  STRUCT
   STAT0 : ARRAY  [0 .. 999 ] OF BOOL ;
  END_STRUCT ;
BEGIN
   STAT0[0] := FALSE;
   STAT0[1] := FALSE;
   STAT0[2] := FALSE;
   STAT0[3] := FALSE;
   STAT0[4] := FALSE;
   STAT0[5] := FALSE;
   STAT0[6] := FALSE;
   STAT0[7] := FALSE;
   STAT0[8] := FALSE;
   STAT0[9] := FALSE;
   STAT0[10] := FALSE;
   STAT0[11] := FALSE;
   STAT0[12] := FALSE;
   STAT0[13] := FALSE;
   STAT0[14] := FALSE;
   STAT0[15] := FALSE;
   STAT0[16] := FALSE;
   STAT0[17] := FALSE;
   STAT0[18] := FALSE;
   STAT0[19] := FALSE;
   STAT0[20] := FALSE;
   STAT0[21] := FALSE;
   STAT0[22] := FALSE;
   STAT0[23] := FALSE;
   STAT0[24] := FALSE;
   STAT0[25] := FALSE;
   STAT0[26] := FALSE;
   STAT0[27] := FALSE;
   STAT0[28] := FALSE;
   STAT0[29] := FALSE;
   STAT0[30] := FALSE;
   STAT0[31] := FALSE;
   STAT0[32] := FALSE;
   STAT0[33] := FALSE;
   STAT0[34] := FALSE;
   STAT0[35] := FALSE;
   STAT0[36] := FALSE;
   STAT0[37] := FALSE;
   STAT0[38] := FALSE;
   STAT0[39] := FALSE;
   STAT0[40] := FALSE;
   STAT0[41] := FALSE;
   STAT0[42] := FALSE;
   STAT0[43] := FALSE;
   STAT0[44] := FALSE;
   STAT0[45] := FALSE;
   STAT0[46] := FALSE;
   STAT0[47] := FALSE;
   STAT0[48] := FALSE;
   STAT0[49] := FALSE;
   STAT0[50] := FALSE;
   STAT0[51] := FALSE;
   STAT0[52] := FALSE;
   STAT0[53] := FALSE;
   STAT0[54] := FALSE;
   STAT0[55] := FALSE;
   STAT0[56] := FALSE;
   STAT0[57] := FALSE;
   STAT0[58] := FALSE;
   STAT0[59] := FALSE;
   STAT0[60] := FALSE;
   STAT0[61] := FALSE;
   STAT0[62] := FALSE;
   STAT0[63] := FALSE;
   STAT0[64] := FALSE;
   STAT0[65] := FALSE;
   STAT0[66] := FALSE;
   STAT0[67] := FALSE;
   STAT0[68] := FALSE;
   STAT0[69] := FALSE;
   STAT0[70] := FALSE;
   STAT0[71] := FALSE;
   STAT0[72] := FALSE;
   STAT0[73] := FALSE;
   STAT0[74] := FALSE;
   STAT0[75] := FALSE;
   STAT0[76] := FALSE;
   STAT0[77] := FALSE;
   STAT0[78] := FALSE;
   STAT0[79] := FALSE;
   STAT0[80] := FALSE;
   STAT0[81] := FALSE;
   STAT0[82] := FALSE;
   STAT0[83] := FALSE;
   STAT0[84] := FALSE;
   STAT0[85] := FALSE;
   STAT0[86] := FALSE;
   STAT0[87] := FALSE;
   STAT0[88] := FALSE;
   STAT0[89] := FALSE;
   STAT0[90] := FALSE;
   STAT0[91] := FALSE;
   STAT0[92] := FALSE;
   STAT0[93] := FALSE;
   STAT0[94] := FALSE;
   STAT0[95] := FALSE;
   STAT0[96] := FALSE;
   STAT0[97] := FALSE;
   STAT0[98] := FALSE;
   STAT0[99] := FALSE;
   STAT0[100] := FALSE;
   STAT0[101] := FALSE;
   STAT0[102] := FALSE;
   STAT0[103] := FALSE;
   STAT0[104] := FALSE;
   STAT0[105] := FALSE;
   STAT0[106] := FALSE;
   STAT0[107] := FALSE;
   STAT0[108] := FALSE;
   STAT0[109] := FALSE;
   STAT0[110] := FALSE;
   STAT0[111] := FALSE;
   STAT0[112] := FALSE;
   STAT0[113] := FALSE;
   STAT0[114] := FALSE;
   STAT0[115] := FALSE;
   STAT0[116] := FALSE;
   STAT0[117] := FALSE;
   STAT0[118] := FALSE;
   STAT0[119] := FALSE;
   STAT0[120] := FALSE;
   STAT0[121] := FALSE;
   STAT0[122] := FALSE;
   STAT0[123] := FALSE;
   STAT0[124] := FALSE;
   STAT0[125] := FALSE;
   STAT0[126] := FALSE;
   STAT0[127] := FALSE;
   STAT0[128] := FALSE;
   STAT0[129] := FALSE;
   STAT0[130] := FALSE;
   STAT0[131] := FALSE;
   STAT0[132] := FALSE;
   STAT0[133] := FALSE;
   STAT0[134] := FALSE;
   STAT0[135] := FALSE;
   STAT0[136] := FALSE;
   STAT0[137] := FALSE;
   STAT0[138] := FALSE;
   STAT0[139] := FALSE;
   STAT0[140] := FALSE;
   STAT0[141] := FALSE;
   STAT0[142] := FALSE;
   STAT0[143] := FALSE;
   STAT0[144] := FALSE;
   STAT0[145] := FALSE;
   STAT0[146] := FALSE;
   STAT0[147] := FALSE;
   STAT0[148] := FALSE;
   STAT0[149] := FALSE;
   STAT0[150] := FALSE;
   STAT0[151] := FALSE;
   STAT0[152] := FALSE;
   STAT0[153] := FALSE;
   STAT0[154] := FALSE;
   STAT0[155] := FALSE;
   STAT0[156] := FALSE;
   STAT0[157] := FALSE;
   STAT0[158] := FALSE;
   STAT0[159] := FALSE;
   STAT0[160] := FALSE;
   STAT0[161] := FALSE;
   STAT0[162] := FALSE;
   STAT0[163] := FALSE;
   STAT0[164] := FALSE;
   STAT0[165] := FALSE;
   STAT0[166] := FALSE;
   STAT0[167] := FALSE;
   STAT0[168] := FALSE;
   STAT0[169] := FALSE;
   STAT0[170] := FALSE;
   STAT0[171] := FALSE;
   STAT0[172] := FALSE;
   STAT0[173] := FALSE;
   STAT0[174] := FALSE;
   STAT0[175] := FALSE;
   STAT0[176] := FALSE;
   STAT0[177] := FALSE;
   STAT0[178] := FALSE;
   STAT0[179] := FALSE;
   STAT0[180] := FALSE;
   STAT0[181] := FALSE;
   STAT0[182] := FALSE;
   STAT0[183] := FALSE;
   STAT0[184] := FALSE;
   STAT0[185] := FALSE;
   STAT0[186] := FALSE;
   STAT0[187] := FALSE;
   STAT0[188] := FALSE;
   STAT0[189] := FALSE;
   STAT0[190] := FALSE;
   STAT0[191] := FALSE;
   STAT0[192] := FALSE;
   STAT0[193] := FALSE;
   STAT0[194] := FALSE;
   STAT0[195] := FALSE;
   STAT0[196] := FALSE;
   STAT0[197] := FALSE;
   STAT0[198] := FALSE;
   STAT0[199] := FALSE;
   STAT0[200] := FALSE;
   STAT0[201] := FALSE;
   STAT0[202] := FALSE;
   STAT0[203] := FALSE;
   STAT0[204] := FALSE;
   STAT0[205] := FALSE;
   STAT0[206] := FALSE;
   STAT0[207] := FALSE;
   STAT0[208] := FALSE;
   STAT0[209] := FALSE;
   STAT0[210] := FALSE;
   STAT0[211] := FALSE;
   STAT0[212] := FALSE;
   STAT0[213] := FALSE;
   STAT0[214] := FALSE;
   STAT0[215] := FALSE;
   STAT0[216] := FALSE;
   STAT0[217] := FALSE;
   STAT0[218] := FALSE;
   STAT0[219] := FALSE;
   STAT0[220] := FALSE;
   STAT0[221] := FALSE;
   STAT0[222] := FALSE;
   STAT0[223] := FALSE;
   STAT0[224] := FALSE;
   STAT0[225] := FALSE;
   STAT0[226] := FALSE;
   STAT0[227] := FALSE;
   STAT0[228] := FALSE;
   STAT0[229] := FALSE;
   STAT0[230] := FALSE;
   STAT0[231] := FALSE;
   STAT0[232] := FALSE;
   STAT0[233] := FALSE;
   STAT0[234] := FALSE;
   STAT0[235] := FALSE;
   STAT0[236] := FALSE;
   STAT0[237] := FALSE;
   STAT0[238] := FALSE;
   STAT0[239] := FALSE;
   STAT0[240] := FALSE;
   STAT0[241] := FALSE;
   STAT0[242] := FALSE;
   STAT0[243] := FALSE;
   STAT0[244] := FALSE;
   STAT0[245] := FALSE;
   STAT0[246] := FALSE;
   STAT0[247] := FALSE;
   STAT0[248] := FALSE;
   STAT0[249] := FALSE;
   STAT0[250] := FALSE;
   STAT0[251] := FALSE;
   STAT0[252] := FALSE;
   STAT0[253] := FALSE;
   STAT0[254] := FALSE;
   STAT0[255] := FALSE;
   STAT0[256] := FALSE;
   STAT0[257] := FALSE;
   STAT0[258] := FALSE;
   STAT0[259] := FALSE;
   STAT0[260] := FALSE;
   STAT0[261] := FALSE;
   STAT0[262] := FALSE;
   STAT0[263] := FALSE;
   STAT0[264] := FALSE;
   STAT0[265] := FALSE;
   STAT0[266] := FALSE;
   STAT0[267] := FALSE;
   STAT0[268] := FALSE;
   STAT0[269] := FALSE;
   STAT0[270] := FALSE;
   STAT0[271] := FALSE;
   STAT0[272] := FALSE;
   STAT0[273] := FALSE;
   STAT0[274] := FALSE;
   STAT0[275] := FALSE;
   STAT0[276] := FALSE;
   STAT0[277] := FALSE;
   STAT0[278] := FALSE;
   STAT0[279] := FALSE;
   STAT0[280] := FALSE;
   STAT0[281] := FALSE;
   STAT0[282] := FALSE;
   STAT0[283] := FALSE;
   STAT0[284] := FALSE;
   STAT0[285] := FALSE;
   STAT0[286] := FALSE;
   STAT0[287] := FALSE;
   STAT0[288] := FALSE;
   STAT0[289] := FALSE;
   STAT0[290] := FALSE;
   STAT0[291] := FALSE;
   STAT0[292] := FALSE;
   STAT0[293] := FALSE;
   STAT0[294] := FALSE;
   STAT0[295] := FALSE;
   STAT0[296] := FALSE;
   STAT0[297] := FALSE;
   STAT0[298] := FALSE;
   STAT0[299] := FALSE;
   STAT0[300] := FALSE;
   STAT0[301] := FALSE;
   STAT0[302] := FALSE;
   STAT0[303] := FALSE;
   STAT0[304] := FALSE;
   STAT0[305] := FALSE;
   STAT0[306] := FALSE;
   STAT0[307] := FALSE;
   STAT0[308] := FALSE;
   STAT0[309] := FALSE;
   STAT0[310] := FALSE;
   STAT0[311] := FALSE;
   STAT0[312] := FALSE;
   STAT0[313] := FALSE;
   STAT0[314] := FALSE;
   STAT0[315] := FALSE;
   STAT0[316] := FALSE;
   STAT0[317] := FALSE;
   STAT0[318] := FALSE;
   STAT0[319] := FALSE;
   STAT0[320] := FALSE;
   STAT0[321] := FALSE;
   STAT0[322] := FALSE;
   STAT0[323] := FALSE;
   STAT0[324] := FALSE;
   STAT0[325] := FALSE;
   STAT0[326] := FALSE;
   STAT0[327] := FALSE;
   STAT0[328] := FALSE;
   STAT0[329] := FALSE;
   STAT0[330] := FALSE;
   STAT0[331] := FALSE;
   STAT0[332] := FALSE;
   STAT0[333] := FALSE;
   STAT0[334] := FALSE;
   STAT0[335] := FALSE;
   STAT0[336] := FALSE;
   STAT0[337] := FALSE;
   STAT0[338] := FALSE;
   STAT0[339] := FALSE;
   STAT0[340] := FALSE;
   STAT0[341] := FALSE;
   STAT0[342] := FALSE;
   STAT0[343] := FALSE;
   STAT0[344] := FALSE;
   STAT0[345] := FALSE;
   STAT0[346] := FALSE;
   STAT0[347] := FALSE;
   STAT0[348] := FALSE;
   STAT0[349] := FALSE;
   STAT0[350] := FALSE;
   STAT0[351] := FALSE;
   STAT0[352] := FALSE;
   STAT0[353] := FALSE;
   STAT0[354] := FALSE;
   STAT0[355] := FALSE;
   STAT0[356] := FALSE;
   STAT0[357] := FALSE;
   STAT0[358] := FALSE;
   STAT0[359] := FALSE;
   STAT0[360] := FALSE;
   STAT0[361] := FALSE;
   STAT0[362] := FALSE;
   STAT0[363] := FALSE;
   STAT0[364] := FALSE;
   STAT0[365] := FALSE;
   STAT0[366] := FALSE;
   STAT0[367] := FALSE;
   STAT0[368] := FALSE;
   STAT0[369] := FALSE;
   STAT0[370] := FALSE;
   STAT0[371] := FALSE;
   STAT0[372] := FALSE;
   STAT0[373] := FALSE;
   STAT0[374] := FALSE;
   STAT0[375] := FALSE;
   STAT0[376] := FALSE;
   STAT0[377] := FALSE;
   STAT0[378] := FALSE;
   STAT0[379] := FALSE;
   STAT0[380] := FALSE;
   STAT0[381] := FALSE;
   STAT0[382] := FALSE;
   STAT0[383] := FALSE;
   STAT0[384] := FALSE;
   STAT0[385] := FALSE;
   STAT0[386] := FALSE;
   STAT0[387] := FALSE;
   STAT0[388] := FALSE;
   STAT0[389] := FALSE;
   STAT0[390] := FALSE;
   STAT0[391] := FALSE;
   STAT0[392] := FALSE;
   STAT0[393] := FALSE;
   STAT0[394] := FALSE;
   STAT0[395] := FALSE;
   STAT0[396] := FALSE;
   STAT0[397] := FALSE;
   STAT0[398] := FALSE;
   STAT0[399] := FALSE;
   STAT0[400] := FALSE;
   STAT0[401] := FALSE;
   STAT0[402] := FALSE;
   STAT0[403] := FALSE;
   STAT0[404] := FALSE;
   STAT0[405] := FALSE;
   STAT0[406] := FALSE;
   STAT0[407] := FALSE;
   STAT0[408] := FALSE;
   STAT0[409] := FALSE;
   STAT0[410] := FALSE;
   STAT0[411] := FALSE;
   STAT0[412] := FALSE;
   STAT0[413] := FALSE;
   STAT0[414] := FALSE;
   STAT0[415] := FALSE;
   STAT0[416] := FALSE;
   STAT0[417] := FALSE;
   STAT0[418] := FALSE;
   STAT0[419] := FALSE;
   STAT0[420] := FALSE;
   STAT0[421] := FALSE;
   STAT0[422] := FALSE;
   STAT0[423] := FALSE;
   STAT0[424] := FALSE;
   STAT0[425] := FALSE;
   STAT0[426] := FALSE;
   STAT0[427] := FALSE;
   STAT0[428] := FALSE;
   STAT0[429] := FALSE;
   STAT0[430] := FALSE;
   STAT0[431] := FALSE;
   STAT0[432] := FALSE;
   STAT0[433] := FALSE;
   STAT0[434] := FALSE;
   STAT0[435] := FALSE;
   STAT0[436] := FALSE;
   STAT0[437] := FALSE;
   STAT0[438] := FALSE;
   STAT0[439] := FALSE;
   STAT0[440] := FALSE;
   STAT0[441] := FALSE;
   STAT0[442] := FALSE;
   STAT0[443] := FALSE;
   STAT0[444] := FALSE;
   STAT0[445] := FALSE;
   STAT0[446] := FALSE;
   STAT0[447] := FALSE;
   STAT0[448] := FALSE;
   STAT0[449] := FALSE;
   STAT0[450] := FALSE;
   STAT0[451] := FALSE;
   STAT0[452] := FALSE;
   STAT0[453] := FALSE;
   STAT0[454] := FALSE;
   STAT0[455] := FALSE;
   STAT0[456] := FALSE;
   STAT0[457] := FALSE;
   STAT0[458] := FALSE;
   STAT0[459] := FALSE;
   STAT0[460] := FALSE;
   STAT0[461] := FALSE;
   STAT0[462] := FALSE;
   STAT0[463] := FALSE;
   STAT0[464] := FALSE;
   STAT0[465] := FALSE;
   STAT0[466] := FALSE;
   STAT0[467] := FALSE;
   STAT0[468] := FALSE;
   STAT0[469] := FALSE;
   STAT0[470] := FALSE;
   STAT0[471] := FALSE;
   STAT0[472] := FALSE;
   STAT0[473] := FALSE;
   STAT0[474] := FALSE;
   STAT0[475] := FALSE;
   STAT0[476] := FALSE;
   STAT0[477] := FALSE;
   STAT0[478] := FALSE;
   STAT0[479] := FALSE;
   STAT0[480] := FALSE;
   STAT0[481] := FALSE;
   STAT0[482] := FALSE;
   STAT0[483] := FALSE;
   STAT0[484] := FALSE;
   STAT0[485] := FALSE;
   STAT0[486] := FALSE;
   STAT0[487] := FALSE;
   STAT0[488] := FALSE;
   STAT0[489] := FALSE;
   STAT0[490] := FALSE;
   STAT0[491] := FALSE;
   STAT0[492] := FALSE;
   STAT0[493] := FALSE;
   STAT0[494] := FALSE;
   STAT0[495] := FALSE;
   STAT0[496] := FALSE;
   STAT0[497] := FALSE;
   STAT0[498] := FALSE;
   STAT0[499] := FALSE;
   STAT0[500] := FALSE;
   STAT0[501] := FALSE;
   STAT0[502] := FALSE;
   STAT0[503] := FALSE;
   STAT0[504] := FALSE;
   STAT0[505] := FALSE;
   STAT0[506] := FALSE;
   STAT0[507] := FALSE;
   STAT0[508] := FALSE;
   STAT0[509] := FALSE;
   STAT0[510] := FALSE;
   STAT0[511] := FALSE;
   STAT0[512] := FALSE;
   STAT0[513] := FALSE;
   STAT0[514] := FALSE;
   STAT0[515] := FALSE;
   STAT0[516] := FALSE;
   STAT0[517] := FALSE;
   STAT0[518] := FALSE;
   STAT0[519] := FALSE;
   STAT0[520] := FALSE;
   STAT0[521] := FALSE;
   STAT0[522] := FALSE;
   STAT0[523] := FALSE;
   STAT0[524] := FALSE;
   STAT0[525] := FALSE;
   STAT0[526] := FALSE;
   STAT0[527] := FALSE;
   STAT0[528] := FALSE;
   STAT0[529] := FALSE;
   STAT0[530] := FALSE;
   STAT0[531] := FALSE;
   STAT0[532] := FALSE;
   STAT0[533] := FALSE;
   STAT0[534] := FALSE;
   STAT0[535] := FALSE;
   STAT0[536] := FALSE;
   STAT0[537] := FALSE;
   STAT0[538] := FALSE;
   STAT0[539] := FALSE;
   STAT0[540] := FALSE;
   STAT0[541] := FALSE;
   STAT0[542] := FALSE;
   STAT0[543] := FALSE;
   STAT0[544] := FALSE;
   STAT0[545] := FALSE;
   STAT0[546] := FALSE;
   STAT0[547] := FALSE;
   STAT0[548] := FALSE;
   STAT0[549] := FALSE;
   STAT0[550] := FALSE;
   STAT0[551] := FALSE;
   STAT0[552] := FALSE;
   STAT0[553] := FALSE;
   STAT0[554] := FALSE;
   STAT0[555] := FALSE;
   STAT0[556] := FALSE;
   STAT0[557] := FALSE;
   STAT0[558] := FALSE;
   STAT0[559] := FALSE;
   STAT0[560] := FALSE;
   STAT0[561] := FALSE;
   STAT0[562] := FALSE;
   STAT0[563] := FALSE;
   STAT0[564] := FALSE;
   STAT0[565] := FALSE;
   STAT0[566] := FALSE;
   STAT0[567] := FALSE;
   STAT0[568] := FALSE;
   STAT0[569] := FALSE;
   STAT0[570] := FALSE;
   STAT0[571] := FALSE;
   STAT0[572] := FALSE;
   STAT0[573] := FALSE;
   STAT0[574] := FALSE;
   STAT0[575] := FALSE;
   STAT0[576] := FALSE;
   STAT0[577] := FALSE;
   STAT0[578] := FALSE;
   STAT0[579] := FALSE;
   STAT0[580] := FALSE;
   STAT0[581] := FALSE;
   STAT0[582] := FALSE;
   STAT0[583] := FALSE;
   STAT0[584] := FALSE;
   STAT0[585] := FALSE;
   STAT0[586] := FALSE;
   STAT0[587] := FALSE;
   STAT0[588] := FALSE;
   STAT0[589] := FALSE;
   STAT0[590] := FALSE;
   STAT0[591] := FALSE;
   STAT0[592] := FALSE;
   STAT0[593] := FALSE;
   STAT0[594] := FALSE;
   STAT0[595] := FALSE;
   STAT0[596] := FALSE;
   STAT0[597] := FALSE;
   STAT0[598] := FALSE;
   STAT0[599] := FALSE;
   STAT0[600] := FALSE;
   STAT0[601] := FALSE;
   STAT0[602] := FALSE;
   STAT0[603] := FALSE;
   STAT0[604] := FALSE;
   STAT0[605] := FALSE;
   STAT0[606] := FALSE;
   STAT0[607] := FALSE;
   STAT0[608] := FALSE;
   STAT0[609] := FALSE;
   STAT0[610] := FALSE;
   STAT0[611] := FALSE;
   STAT0[612] := FALSE;
   STAT0[613] := FALSE;
   STAT0[614] := FALSE;
   STAT0[615] := FALSE;
   STAT0[616] := FALSE;
   STAT0[617] := FALSE;
   STAT0[618] := FALSE;
   STAT0[619] := FALSE;
   STAT0[620] := FALSE;
   STAT0[621] := FALSE;
   STAT0[622] := FALSE;
   STAT0[623] := FALSE;
   STAT0[624] := FALSE;
   STAT0[625] := FALSE;
   STAT0[626] := FALSE;
   STAT0[627] := FALSE;
   STAT0[628] := FALSE;
   STAT0[629] := FALSE;
   STAT0[630] := FALSE;
   STAT0[631] := FALSE;
   STAT0[632] := FALSE;
   STAT0[633] := FALSE;
   STAT0[634] := FALSE;
   STAT0[635] := FALSE;
   STAT0[636] := FALSE;
   STAT0[637] := FALSE;
   STAT0[638] := FALSE;
   STAT0[639] := FALSE;
   STAT0[640] := FALSE;
   STAT0[641] := FALSE;
   STAT0[642] := FALSE;
   STAT0[643] := FALSE;
   STAT0[644] := FALSE;
   STAT0[645] := FALSE;
   STAT0[646] := FALSE;
   STAT0[647] := FALSE;
   STAT0[648] := FALSE;
   STAT0[649] := FALSE;
   STAT0[650] := FALSE;
   STAT0[651] := FALSE;
   STAT0[652] := FALSE;
   STAT0[653] := FALSE;
   STAT0[654] := FALSE;
   STAT0[655] := FALSE;
   STAT0[656] := FALSE;
   STAT0[657] := FALSE;
   STAT0[658] := FALSE;
   STAT0[659] := FALSE;
   STAT0[660] := FALSE;
   STAT0[661] := FALSE;
   STAT0[662] := FALSE;
   STAT0[663] := FALSE;
   STAT0[664] := FALSE;
   STAT0[665] := FALSE;
   STAT0[666] := FALSE;
   STAT0[667] := FALSE;
   STAT0[668] := FALSE;
   STAT0[669] := FALSE;
   STAT0[670] := FALSE;
   STAT0[671] := FALSE;
   STAT0[672] := FALSE;
   STAT0[673] := FALSE;
   STAT0[674] := FALSE;
   STAT0[675] := FALSE;
   STAT0[676] := FALSE;
   STAT0[677] := FALSE;
   STAT0[678] := FALSE;
   STAT0[679] := FALSE;
   STAT0[680] := FALSE;
   STAT0[681] := FALSE;
   STAT0[682] := FALSE;
   STAT0[683] := FALSE;
   STAT0[684] := FALSE;
   STAT0[685] := FALSE;
   STAT0[686] := FALSE;
   STAT0[687] := FALSE;
   STAT0[688] := FALSE;
   STAT0[689] := FALSE;
   STAT0[690] := FALSE;
   STAT0[691] := FALSE;
   STAT0[692] := FALSE;
   STAT0[693] := FALSE;
   STAT0[694] := FALSE;
   STAT0[695] := FALSE;
   STAT0[696] := FALSE;
   STAT0[697] := FALSE;
   STAT0[698] := FALSE;
   STAT0[699] := FALSE;
   STAT0[700] := FALSE;
   STAT0[701] := FALSE;
   STAT0[702] := FALSE;
   STAT0[703] := FALSE;
   STAT0[704] := FALSE;
   STAT0[705] := FALSE;
   STAT0[706] := FALSE;
   STAT0[707] := FALSE;
   STAT0[708] := FALSE;
   STAT0[709] := FALSE;
   STAT0[710] := FALSE;
   STAT0[711] := FALSE;
   STAT0[712] := FALSE;
   STAT0[713] := FALSE;
   STAT0[714] := FALSE;
   STAT0[715] := FALSE;
   STAT0[716] := FALSE;
   STAT0[717] := FALSE;
   STAT0[718] := FALSE;
   STAT0[719] := FALSE;
   STAT0[720] := FALSE;
   STAT0[721] := FALSE;
   STAT0[722] := FALSE;
   STAT0[723] := FALSE;
   STAT0[724] := FALSE;
   STAT0[725] := FALSE;
   STAT0[726] := FALSE;
   STAT0[727] := FALSE;
   STAT0[728] := FALSE;
   STAT0[729] := FALSE;
   STAT0[730] := FALSE;
   STAT0[731] := FALSE;
   STAT0[732] := FALSE;
   STAT0[733] := FALSE;
   STAT0[734] := FALSE;
   STAT0[735] := FALSE;
   STAT0[736] := FALSE;
   STAT0[737] := FALSE;
   STAT0[738] := FALSE;
   STAT0[739] := FALSE;
   STAT0[740] := FALSE;
   STAT0[741] := FALSE;
   STAT0[742] := FALSE;
   STAT0[743] := FALSE;
   STAT0[744] := FALSE;
   STAT0[745] := FALSE;
   STAT0[746] := FALSE;
   STAT0[747] := FALSE;
   STAT0[748] := FALSE;
   STAT0[749] := FALSE;
   STAT0[750] := FALSE;
   STAT0[751] := FALSE;
   STAT0[752] := FALSE;
   STAT0[753] := FALSE;
   STAT0[754] := FALSE;
   STAT0[755] := FALSE;
   STAT0[756] := FALSE;
   STAT0[757] := FALSE;
   STAT0[758] := FALSE;
   STAT0[759] := FALSE;
   STAT0[760] := FALSE;
   STAT0[761] := FALSE;
   STAT0[762] := FALSE;
   STAT0[763] := FALSE;
   STAT0[764] := FALSE;
   STAT0[765] := FALSE;
   STAT0[766] := FALSE;
   STAT0[767] := FALSE;
   STAT0[768] := FALSE;
   STAT0[769] := FALSE;
   STAT0[770] := FALSE;
   STAT0[771] := FALSE;
   STAT0[772] := FALSE;
   STAT0[773] := FALSE;
   STAT0[774] := FALSE;
   STAT0[775] := FALSE;
   STAT0[776] := FALSE;
   STAT0[777] := FALSE;
   STAT0[778] := FALSE;
   STAT0[779] := FALSE;
   STAT0[780] := FALSE;
   STAT0[781] := FALSE;
   STAT0[782] := FALSE;
   STAT0[783] := FALSE;
   STAT0[784] := FALSE;
   STAT0[785] := FALSE;
   STAT0[786] := FALSE;
   STAT0[787] := FALSE;
   STAT0[788] := FALSE;
   STAT0[789] := FALSE;
   STAT0[790] := FALSE;
   STAT0[791] := FALSE;
   STAT0[792] := FALSE;
   STAT0[793] := FALSE;
   STAT0[794] := FALSE;
   STAT0[795] := FALSE;
   STAT0[796] := FALSE;
   STAT0[797] := FALSE;
   STAT0[798] := FALSE;
   STAT0[799] := FALSE;
   STAT0[800] := FALSE;
   STAT0[801] := FALSE;
   STAT0[802] := FALSE;
   STAT0[803] := FALSE;
   STAT0[804] := FALSE;
   STAT0[805] := FALSE;
   STAT0[806] := FALSE;
   STAT0[807] := FALSE;
   STAT0[808] := FALSE;
   STAT0[809] := FALSE;
   STAT0[810] := FALSE;
   STAT0[811] := FALSE;
   STAT0[812] := FALSE;
   STAT0[813] := FALSE;
   STAT0[814] := FALSE;
   STAT0[815] := FALSE;
   STAT0[816] := FALSE;
   STAT0[817] := FALSE;
   STAT0[818] := FALSE;
   STAT0[819] := FALSE;
   STAT0[820] := FALSE;
   STAT0[821] := FALSE;
   STAT0[822] := FALSE;
   STAT0[823] := FALSE;
   STAT0[824] := FALSE;
   STAT0[825] := FALSE;
   STAT0[826] := FALSE;
   STAT0[827] := FALSE;
   STAT0[828] := FALSE;
   STAT0[829] := FALSE;
   STAT0[830] := FALSE;
   STAT0[831] := FALSE;
   STAT0[832] := FALSE;
   STAT0[833] := FALSE;
   STAT0[834] := FALSE;
   STAT0[835] := FALSE;
   STAT0[836] := FALSE;
   STAT0[837] := FALSE;
   STAT0[838] := FALSE;
   STAT0[839] := FALSE;
   STAT0[840] := FALSE;
   STAT0[841] := FALSE;
   STAT0[842] := FALSE;
   STAT0[843] := FALSE;
   STAT0[844] := FALSE;
   STAT0[845] := FALSE;
   STAT0[846] := FALSE;
   STAT0[847] := FALSE;
   STAT0[848] := FALSE;
   STAT0[849] := FALSE;
   STAT0[850] := FALSE;
   STAT0[851] := FALSE;
   STAT0[852] := FALSE;
   STAT0[853] := FALSE;
   STAT0[854] := FALSE;
   STAT0[855] := FALSE;
   STAT0[856] := FALSE;
   STAT0[857] := FALSE;
   STAT0[858] := FALSE;
   STAT0[859] := FALSE;
   STAT0[860] := FALSE;
   STAT0[861] := FALSE;
   STAT0[862] := FALSE;
   STAT0[863] := FALSE;
   STAT0[864] := FALSE;
   STAT0[865] := FALSE;
   STAT0[866] := FALSE;
   STAT0[867] := FALSE;
   STAT0[868] := FALSE;
   STAT0[869] := FALSE;
   STAT0[870] := FALSE;
   STAT0[871] := FALSE;
   STAT0[872] := FALSE;
   STAT0[873] := FALSE;
   STAT0[874] := FALSE;
   STAT0[875] := FALSE;
   STAT0[876] := FALSE;
   STAT0[877] := FALSE;
   STAT0[878] := FALSE;
   STAT0[879] := FALSE;
   STAT0[880] := FALSE;
   STAT0[881] := FALSE;
   STAT0[882] := FALSE;
   STAT0[883] := FALSE;
   STAT0[884] := FALSE;
   STAT0[885] := FALSE;
   STAT0[886] := FALSE;
   STAT0[887] := FALSE;
   STAT0[888] := FALSE;
   STAT0[889] := FALSE;
   STAT0[890] := FALSE;
   STAT0[891] := FALSE;
   STAT0[892] := FALSE;
   STAT0[893] := FALSE;
   STAT0[894] := FALSE;
   STAT0[895] := FALSE;
   STAT0[896] := FALSE;
   STAT0[897] := FALSE;
   STAT0[898] := FALSE;
   STAT0[899] := FALSE;
   STAT0[900] := FALSE;
   STAT0[901] := FALSE;
   STAT0[902] := FALSE;
   STAT0[903] := FALSE;
   STAT0[904] := FALSE;
   STAT0[905] := FALSE;
   STAT0[906] := FALSE;
   STAT0[907] := FALSE;
   STAT0[908] := FALSE;
   STAT0[909] := FALSE;
   STAT0[910] := FALSE;
   STAT0[911] := FALSE;
   STAT0[912] := FALSE;
   STAT0[913] := FALSE;
   STAT0[914] := FALSE;
   STAT0[915] := FALSE;
   STAT0[916] := FALSE;
   STAT0[917] := FALSE;
   STAT0[918] := FALSE;
   STAT0[919] := FALSE;
   STAT0[920] := FALSE;
   STAT0[921] := FALSE;
   STAT0[922] := FALSE;
   STAT0[923] := FALSE;
   STAT0[924] := FALSE;
   STAT0[925] := FALSE;
   STAT0[926] := FALSE;
   STAT0[927] := FALSE;
   STAT0[928] := FALSE;
   STAT0[929] := FALSE;
   STAT0[930] := FALSE;
   STAT0[931] := FALSE;
   STAT0[932] := FALSE;
   STAT0[933] := FALSE;
   STAT0[934] := FALSE;
   STAT0[935] := FALSE;
   STAT0[936] := FALSE;
   STAT0[937] := FALSE;
   STAT0[938] := FALSE;
   STAT0[939] := FALSE;
   STAT0[940] := FALSE;
   STAT0[941] := FALSE;
   STAT0[942] := FALSE;
   STAT0[943] := FALSE;
   STAT0[944] := FALSE;
   STAT0[945] := FALSE;
   STAT0[946] := FALSE;
   STAT0[947] := FALSE;
   STAT0[948] := FALSE;
   STAT0[949] := FALSE;
   STAT0[950] := FALSE;
   STAT0[951] := FALSE;
   STAT0[952] := FALSE;
   STAT0[953] := FALSE;
   STAT0[954] := FALSE;
   STAT0[955] := FALSE;
   STAT0[956] := FALSE;
   STAT0[957] := FALSE;
   STAT0[958] := FALSE;
   STAT0[959] := FALSE;
   STAT0[960] := FALSE;
   STAT0[961] := FALSE;
   STAT0[962] := FALSE;
   STAT0[963] := FALSE;
   STAT0[964] := FALSE;
   STAT0[965] := FALSE;
   STAT0[966] := FALSE;
   STAT0[967] := FALSE;
   STAT0[968] := FALSE;
   STAT0[969] := FALSE;
   STAT0[970] := FALSE;
   STAT0[971] := FALSE;
   STAT0[972] := FALSE;
   STAT0[973] := FALSE;
   STAT0[974] := FALSE;
   STAT0[975] := FALSE;
   STAT0[976] := FALSE;
   STAT0[977] := FALSE;
   STAT0[978] := FALSE;
   STAT0[979] := FALSE;
   STAT0[980] := FALSE;
   STAT0[981] := FALSE;
   STAT0[982] := FALSE;
   STAT0[983] := FALSE;
   STAT0[984] := FALSE;
   STAT0[985] := FALSE;
   STAT0[986] := FALSE;
   STAT0[987] := FALSE;
   STAT0[988] := FALSE;
   STAT0[989] := FALSE;
   STAT0[990] := FALSE;
   STAT0[991] := FALSE;
   STAT0[992] := FALSE;
   STAT0[993] := FALSE;
   STAT0[994] := FALSE;
   STAT0[995] := FALSE;
   STAT0[996] := FALSE;
   STAT0[997] := FALSE;
   STAT0[998] := FALSE;
   STAT0[999] := FALSE;
END_DATA_BLOCK

DATA_BLOCK DB 325
TITLE =
VERSION : 0.1


  STRUCT
   DP_DIAG1 : ARRAY  [1 .. 100 ] OF BYTE ;
   DP_DIAG2 : ARRAY  [1 .. 100 ] OF BYTE ;
   DP_DIAG3 : ARRAY  [1 .. 100 ] OF BYTE ;
   DP_DIAG4 : ARRAY  [1 .. 100 ] OF BYTE ;
   DP_DIAG5 : ARRAY  [1 .. 100 ] OF BYTE ;
   DP_DIAG6 : ARRAY  [1 .. 100 ] OF BYTE ;
   DP_DIAG7 : ARRAY  [1 .. 100 ] OF BYTE ;
   DP_DIAG8 : ARRAY  [1 .. 100 ] OF BYTE ;
   DP_DIAG9 : ARRAY  [1 .. 100 ] OF BYTE ;
   DP_DIAG10 : ARRAY  [1 .. 100 ] OF BYTE ;
  END_STRUCT ;
BEGIN
   DP_DIAG1[1] := B#16#FC;
   DP_DIAG1[2] := B#16#0;
   DP_DIAG1[3] := B#16#8;
   DP_DIAG1[4] := B#16#40;
   DP_DIAG1[5] := B#16#0;
   DP_DIAG1[6] := B#16#0;
   DP_DIAG1[7] := B#16#0;
   DP_DIAG1[8] := B#16#0;
   DP_DIAG1[9] := B#16#0;
   DP_DIAG1[10] := B#16#0;
   DP_DIAG1[11] := B#16#0;
   DP_DIAG1[12] := B#16#0;
   DP_DIAG1[13] := B#16#0;
   DP_DIAG1[14] := B#16#0;
   DP_DIAG1[15] := B#16#0;
   DP_DIAG1[16] := B#16#0;
   DP_DIAG1[17] := B#16#FC;
   DP_DIAG1[18] := B#16#0;
   DP_DIAG1[19] := B#16#8;
   DP_DIAG1[20] := B#16#40;
   DP_DIAG1[21] := B#16#0;
   DP_DIAG1[22] := B#16#0;
   DP_DIAG1[23] := B#16#0;
   DP_DIAG1[24] := B#16#0;
   DP_DIAG1[25] := B#16#0;
   DP_DIAG1[26] := B#16#0;
   DP_DIAG1[27] := B#16#0;
   DP_DIAG1[28] := B#16#0;
   DP_DIAG1[29] := B#16#0;
   DP_DIAG1[30] := B#16#0;
   DP_DIAG1[31] := B#16#0;
   DP_DIAG1[32] := B#16#0;
   DP_DIAG1[33] := B#16#4;
   DP_DIAG1[34] := B#16#0;
   DP_DIAG1[35] := B#16#0;
   DP_DIAG1[36] := B#16#0;
   DP_DIAG1[37] := B#16#0;
   DP_DIAG1[38] := B#16#0;
   DP_DIAG1[39] := B#16#0;
   DP_DIAG1[40] := B#16#0;
   DP_DIAG1[41] := B#16#0;
   DP_DIAG1[42] := B#16#0;
   DP_DIAG1[43] := B#16#0;
   DP_DIAG1[44] := B#16#0;
   DP_DIAG1[45] := B#16#0;
   DP_DIAG1[46] := B#16#0;
   DP_DIAG1[47] := B#16#0;
   DP_DIAG1[48] := B#16#0;
   DP_DIAG1[49] := B#16#0;
   DP_DIAG1[50] := B#16#0;
   DP_DIAG1[51] := B#16#0;
   DP_DIAG1[52] := B#16#0;
   DP_DIAG1[53] := B#16#0;
   DP_DIAG1[54] := B#16#0;
   DP_DIAG1[55] := B#16#0;
   DP_DIAG1[56] := B#16#0;
   DP_DIAG1[57] := B#16#0;
   DP_DIAG1[58] := B#16#0;
   DP_DIAG1[59] := B#16#0;
   DP_DIAG1[60] := B#16#0;
   DP_DIAG1[61] := B#16#0;
   DP_DIAG1[62] := B#16#0;
   DP_DIAG1[63] := B#16#0;
   DP_DIAG1[64] := B#16#0;
   DP_DIAG1[65] := B#16#0;
   DP_DIAG1[66] := B#16#0;
   DP_DIAG1[67] := B#16#4;
   DP_DIAG1[68] := B#16#0;
   DP_DIAG1[69] := B#16#0;
   DP_DIAG1[70] := B#16#0;
   DP_DIAG1[71] := B#16#0;
   DP_DIAG1[72] := B#16#0;
   DP_DIAG1[73] := B#16#0;
   DP_DIAG1[74] := B#16#0;
   DP_DIAG1[75] := B#16#0;
   DP_DIAG1[76] := B#16#0;
   DP_DIAG1[77] := B#16#0;
   DP_DIAG1[78] := B#16#0;
   DP_DIAG1[79] := B#16#0;
   DP_DIAG1[80] := B#16#0;
   DP_DIAG1[81] := B#16#0;
   DP_DIAG1[82] := B#16#0;
   DP_DIAG1[83] := B#16#0;
   DP_DIAG1[84] := B#16#1;
   DP_DIAG1[85] := B#16#0;
   DP_DIAG1[86] := B#16#0;
   DP_DIAG1[87] := B#16#0;
   DP_DIAG1[88] := B#16#0;
   DP_DIAG1[89] := B#16#0;
   DP_DIAG1[90] := B#16#0;
   DP_DIAG1[91] := B#16#0;
   DP_DIAG1[92] := B#16#0;
   DP_DIAG1[93] := B#16#0;
   DP_DIAG1[94] := B#16#0;
   DP_DIAG1[95] := B#16#0;
   DP_DIAG1[96] := B#16#0;
   DP_DIAG1[97] := B#16#0;
   DP_DIAG1[98] := B#16#0;
   DP_DIAG1[99] := B#16#0;
   DP_DIAG1[100] := B#16#0;
   DP_DIAG2[1] := B#16#0;
   DP_DIAG2[2] := B#16#0;
   DP_DIAG2[3] := B#16#0;
   DP_DIAG2[4] := B#16#0;
   DP_DIAG2[5] := B#16#0;
   DP_DIAG2[6] := B#16#0;
   DP_DIAG2[7] := B#16#0;
   DP_DIAG2[8] := B#16#0;
   DP_DIAG2[9] := B#16#0;
   DP_DIAG2[10] := B#16#0;
   DP_DIAG2[11] := B#16#0;
   DP_DIAG2[12] := B#16#0;
   DP_DIAG2[13] := B#16#0;
   DP_DIAG2[14] := B#16#0;
   DP_DIAG2[15] := B#16#0;
   DP_DIAG2[16] := B#16#0;
   DP_DIAG2[17] := B#16#0;
   DP_DIAG2[18] := B#16#0;
   DP_DIAG2[19] := B#16#0;
   DP_DIAG2[20] := B#16#0;
   DP_DIAG2[21] := B#16#0;
   DP_DIAG2[22] := B#16#0;
   DP_DIAG2[23] := B#16#0;
   DP_DIAG2[24] := B#16#0;
   DP_DIAG2[25] := B#16#0;
   DP_DIAG2[26] := B#16#0;
   DP_DIAG2[27] := B#16#0;
   DP_DIAG2[28] := B#16#0;
   DP_DIAG2[29] := B#16#0;
   DP_DIAG2[30] := B#16#0;
   DP_DIAG2[31] := B#16#0;
   DP_DIAG2[32] := B#16#0;
   DP_DIAG2[33] := B#16#0;
   DP_DIAG2[34] := B#16#0;
   DP_DIAG2[35] := B#16#0;
   DP_DIAG2[36] := B#16#0;
   DP_DIAG2[37] := B#16#0;
   DP_DIAG2[38] := B#16#0;
   DP_DIAG2[39] := B#16#0;
   DP_DIAG2[40] := B#16#0;
   DP_DIAG2[41] := B#16#0;
   DP_DIAG2[42] := B#16#0;
   DP_DIAG2[43] := B#16#0;
   DP_DIAG2[44] := B#16#0;
   DP_DIAG2[45] := B#16#0;
   DP_DIAG2[46] := B#16#0;
   DP_DIAG2[47] := B#16#0;
   DP_DIAG2[48] := B#16#0;
   DP_DIAG2[49] := B#16#0;
   DP_DIAG2[50] := B#16#0;
   DP_DIAG2[51] := B#16#0;
   DP_DIAG2[52] := B#16#0;
   DP_DIAG2[53] := B#16#0;
   DP_DIAG2[54] := B#16#0;
   DP_DIAG2[55] := B#16#0;
   DP_DIAG2[56] := B#16#0;
   DP_DIAG2[57] := B#16#0;
   DP_DIAG2[58] := B#16#0;
   DP_DIAG2[59] := B#16#0;
   DP_DIAG2[60] := B#16#0;
   DP_DIAG2[61] := B#16#0;
   DP_DIAG2[62] := B#16#0;
   DP_DIAG2[63] := B#16#0;
   DP_DIAG2[64] := B#16#0;
   DP_DIAG2[65] := B#16#0;
   DP_DIAG2[66] := B#16#0;
   DP_DIAG2[67] := B#16#0;
   DP_DIAG2[68] := B#16#0;
   DP_DIAG2[69] := B#16#0;
   DP_DIAG2[70] := B#16#0;
   DP_DIAG2[71] := B#16#0;
   DP_DIAG2[72] := B#16#0;
   DP_DIAG2[73] := B#16#0;
   DP_DIAG2[74] := B#16#0;
   DP_DIAG2[75] := B#16#0;
   DP_DIAG2[76] := B#16#0;
   DP_DIAG2[77] := B#16#0;
   DP_DIAG2[78] := B#16#0;
   DP_DIAG2[79] := B#16#0;
   DP_DIAG2[80] := B#16#0;
   DP_DIAG2[81] := B#16#0;
   DP_DIAG2[82] := B#16#0;
   DP_DIAG2[83] := B#16#0;
   DP_DIAG2[84] := B#16#0;
   DP_DIAG2[85] := B#16#0;
   DP_DIAG2[86] := B#16#0;
   DP_DIAG2[87] := B#16#0;
   DP_DIAG2[88] := B#16#0;
   DP_DIAG2[89] := B#16#0;
   DP_DIAG2[90] := B#16#0;
   DP_DIAG2[91] := B#16#0;
   DP_DIAG2[92] := B#16#0;
   DP_DIAG2[93] := B#16#0;
   DP_DIAG2[94] := B#16#0;
   DP_DIAG2[95] := B#16#0;
   DP_DIAG2[96] := B#16#0;
   DP_DIAG2[97] := B#16#0;
   DP_DIAG2[98] := B#16#0;
   DP_DIAG2[99] := B#16#0;
   DP_DIAG2[100] := B#16#0;
   DP_DIAG3[1] := B#16#0;
   DP_DIAG3[2] := B#16#0;
   DP_DIAG3[3] := B#16#0;
   DP_DIAG3[4] := B#16#0;
   DP_DIAG3[5] := B#16#0;
   DP_DIAG3[6] := B#16#0;
   DP_DIAG3[7] := B#16#0;
   DP_DIAG3[8] := B#16#0;
   DP_DIAG3[9] := B#16#0;
   DP_DIAG3[10] := B#16#0;
   DP_DIAG3[11] := B#16#0;
   DP_DIAG3[12] := B#16#0;
   DP_DIAG3[13] := B#16#0;
   DP_DIAG3[14] := B#16#0;
   DP_DIAG3[15] := B#16#0;
   DP_DIAG3[16] := B#16#0;
   DP_DIAG3[17] := B#16#0;
   DP_DIAG3[18] := B#16#0;
   DP_DIAG3[19] := B#16#0;
   DP_DIAG3[20] := B#16#0;
   DP_DIAG3[21] := B#16#0;
   DP_DIAG3[22] := B#16#0;
   DP_DIAG3[23] := B#16#0;
   DP_DIAG3[24] := B#16#0;
   DP_DIAG3[25] := B#16#0;
   DP_DIAG3[26] := B#16#0;
   DP_DIAG3[27] := B#16#0;
   DP_DIAG3[28] := B#16#0;
   DP_DIAG3[29] := B#16#0;
   DP_DIAG3[30] := B#16#0;
   DP_DIAG3[31] := B#16#0;
   DP_DIAG3[32] := B#16#0;
   DP_DIAG3[33] := B#16#0;
   DP_DIAG3[34] := B#16#0;
   DP_DIAG3[35] := B#16#0;
   DP_DIAG3[36] := B#16#0;
   DP_DIAG3[37] := B#16#0;
   DP_DIAG3[38] := B#16#0;
   DP_DIAG3[39] := B#16#0;
   DP_DIAG3[40] := B#16#0;
   DP_DIAG3[41] := B#16#0;
   DP_DIAG3[42] := B#16#0;
   DP_DIAG3[43] := B#16#0;
   DP_DIAG3[44] := B#16#0;
   DP_DIAG3[45] := B#16#0;
   DP_DIAG3[46] := B#16#0;
   DP_DIAG3[47] := B#16#0;
   DP_DIAG3[48] := B#16#0;
   DP_DIAG3[49] := B#16#0;
   DP_DIAG3[50] := B#16#0;
   DP_DIAG3[51] := B#16#0;
   DP_DIAG3[52] := B#16#0;
   DP_DIAG3[53] := B#16#0;
   DP_DIAG3[54] := B#16#0;
   DP_DIAG3[55] := B#16#0;
   DP_DIAG3[56] := B#16#0;
   DP_DIAG3[57] := B#16#0;
   DP_DIAG3[58] := B#16#0;
   DP_DIAG3[59] := B#16#0;
   DP_DIAG3[60] := B#16#0;
   DP_DIAG3[61] := B#16#0;
   DP_DIAG3[62] := B#16#0;
   DP_DIAG3[63] := B#16#0;
   DP_DIAG3[64] := B#16#0;
   DP_DIAG3[65] := B#16#0;
   DP_DIAG3[66] := B#16#0;
   DP_DIAG3[67] := B#16#0;
   DP_DIAG3[68] := B#16#0;
   DP_DIAG3[69] := B#16#0;
   DP_DIAG3[70] := B#16#0;
   DP_DIAG3[71] := B#16#0;
   DP_DIAG3[72] := B#16#0;
   DP_DIAG3[73] := B#16#0;
   DP_DIAG3[74] := B#16#0;
   DP_DIAG3[75] := B#16#0;
   DP_DIAG3[76] := B#16#0;
   DP_DIAG3[77] := B#16#0;
   DP_DIAG3[78] := B#16#0;
   DP_DIAG3[79] := B#16#0;
   DP_DIAG3[80] := B#16#0;
   DP_DIAG3[81] := B#16#0;
   DP_DIAG3[82] := B#16#0;
   DP_DIAG3[83] := B#16#0;
   DP_DIAG3[84] := B#16#0;
   DP_DIAG3[85] := B#16#0;
   DP_DIAG3[86] := B#16#0;
   DP_DIAG3[87] := B#16#0;
   DP_DIAG3[88] := B#16#0;
   DP_DIAG3[89] := B#16#0;
   DP_DIAG3[90] := B#16#0;
   DP_DIAG3[91] := B#16#0;
   DP_DIAG3[92] := B#16#0;
   DP_DIAG3[93] := B#16#0;
   DP_DIAG3[94] := B#16#0;
   DP_DIAG3[95] := B#16#0;
   DP_DIAG3[96] := B#16#0;
   DP_DIAG3[97] := B#16#0;
   DP_DIAG3[98] := B#16#0;
   DP_DIAG3[99] := B#16#0;
   DP_DIAG3[100] := B#16#0;
   DP_DIAG4[1] := B#16#0;
   DP_DIAG4[2] := B#16#0;
   DP_DIAG4[3] := B#16#0;
   DP_DIAG4[4] := B#16#0;
   DP_DIAG4[5] := B#16#0;
   DP_DIAG4[6] := B#16#0;
   DP_DIAG4[7] := B#16#0;
   DP_DIAG4[8] := B#16#0;
   DP_DIAG4[9] := B#16#0;
   DP_DIAG4[10] := B#16#0;
   DP_DIAG4[11] := B#16#0;
   DP_DIAG4[12] := B#16#0;
   DP_DIAG4[13] := B#16#0;
   DP_DIAG4[14] := B#16#0;
   DP_DIAG4[15] := B#16#0;
   DP_DIAG4[16] := B#16#0;
   DP_DIAG4[17] := B#16#0;
   DP_DIAG4[18] := B#16#0;
   DP_DIAG4[19] := B#16#0;
   DP_DIAG4[20] := B#16#0;
   DP_DIAG4[21] := B#16#0;
   DP_DIAG4[22] := B#16#0;
   DP_DIAG4[23] := B#16#0;
   DP_DIAG4[24] := B#16#0;
   DP_DIAG4[25] := B#16#0;
   DP_DIAG4[26] := B#16#0;
   DP_DIAG4[27] := B#16#0;
   DP_DIAG4[28] := B#16#0;
   DP_DIAG4[29] := B#16#0;
   DP_DIAG4[30] := B#16#0;
   DP_DIAG4[31] := B#16#0;
   DP_DIAG4[32] := B#16#0;
   DP_DIAG4[33] := B#16#0;
   DP_DIAG4[34] := B#16#0;
   DP_DIAG4[35] := B#16#0;
   DP_DIAG4[36] := B#16#0;
   DP_DIAG4[37] := B#16#0;
   DP_DIAG4[38] := B#16#0;
   DP_DIAG4[39] := B#16#0;
   DP_DIAG4[40] := B#16#0;
   DP_DIAG4[41] := B#16#0;
   DP_DIAG4[42] := B#16#0;
   DP_DIAG4[43] := B#16#0;
   DP_DIAG4[44] := B#16#0;
   DP_DIAG4[45] := B#16#0;
   DP_DIAG4[46] := B#16#0;
   DP_DIAG4[47] := B#16#0;
   DP_DIAG4[48] := B#16#0;
   DP_DIAG4[49] := B#16#0;
   DP_DIAG4[50] := B#16#0;
   DP_DIAG4[51] := B#16#0;
   DP_DIAG4[52] := B#16#0;
   DP_DIAG4[53] := B#16#0;
   DP_DIAG4[54] := B#16#0;
   DP_DIAG4[55] := B#16#0;
   DP_DIAG4[56] := B#16#0;
   DP_DIAG4[57] := B#16#0;
   DP_DIAG4[58] := B#16#0;
   DP_DIAG4[59] := B#16#0;
   DP_DIAG4[60] := B#16#0;
   DP_DIAG4[61] := B#16#0;
   DP_DIAG4[62] := B#16#0;
   DP_DIAG4[63] := B#16#0;
   DP_DIAG4[64] := B#16#0;
   DP_DIAG4[65] := B#16#0;
   DP_DIAG4[66] := B#16#0;
   DP_DIAG4[67] := B#16#0;
   DP_DIAG4[68] := B#16#0;
   DP_DIAG4[69] := B#16#0;
   DP_DIAG4[70] := B#16#0;
   DP_DIAG4[71] := B#16#0;
   DP_DIAG4[72] := B#16#0;
   DP_DIAG4[73] := B#16#0;
   DP_DIAG4[74] := B#16#0;
   DP_DIAG4[75] := B#16#0;
   DP_DIAG4[76] := B#16#0;
   DP_DIAG4[77] := B#16#0;
   DP_DIAG4[78] := B#16#0;
   DP_DIAG4[79] := B#16#0;
   DP_DIAG4[80] := B#16#0;
   DP_DIAG4[81] := B#16#0;
   DP_DIAG4[82] := B#16#0;
   DP_DIAG4[83] := B#16#0;
   DP_DIAG4[84] := B#16#0;
   DP_DIAG4[85] := B#16#0;
   DP_DIAG4[86] := B#16#0;
   DP_DIAG4[87] := B#16#0;
   DP_DIAG4[88] := B#16#0;
   DP_DIAG4[89] := B#16#0;
   DP_DIAG4[90] := B#16#0;
   DP_DIAG4[91] := B#16#0;
   DP_DIAG4[92] := B#16#0;
   DP_DIAG4[93] := B#16#0;
   DP_DIAG4[94] := B#16#0;
   DP_DIAG4[95] := B#16#0;
   DP_DIAG4[96] := B#16#0;
   DP_DIAG4[97] := B#16#0;
   DP_DIAG4[98] := B#16#0;
   DP_DIAG4[99] := B#16#0;
   DP_DIAG4[100] := B#16#0;
   DP_DIAG5[1] := B#16#0;
   DP_DIAG5[2] := B#16#0;
   DP_DIAG5[3] := B#16#0;
   DP_DIAG5[4] := B#16#0;
   DP_DIAG5[5] := B#16#0;
   DP_DIAG5[6] := B#16#0;
   DP_DIAG5[7] := B#16#0;
   DP_DIAG5[8] := B#16#0;
   DP_DIAG5[9] := B#16#0;
   DP_DIAG5[10] := B#16#0;
   DP_DIAG5[11] := B#16#0;
   DP_DIAG5[12] := B#16#0;
   DP_DIAG5[13] := B#16#0;
   DP_DIAG5[14] := B#16#0;
   DP_DIAG5[15] := B#16#0;
   DP_DIAG5[16] := B#16#0;
   DP_DIAG5[17] := B#16#0;
   DP_DIAG5[18] := B#16#0;
   DP_DIAG5[19] := B#16#0;
   DP_DIAG5[20] := B#16#0;
   DP_DIAG5[21] := B#16#0;
   DP_DIAG5[22] := B#16#0;
   DP_DIAG5[23] := B#16#0;
   DP_DIAG5[24] := B#16#0;
   DP_DIAG5[25] := B#16#0;
   DP_DIAG5[26] := B#16#0;
   DP_DIAG5[27] := B#16#0;
   DP_DIAG5[28] := B#16#0;
   DP_DIAG5[29] := B#16#0;
   DP_DIAG5[30] := B#16#0;
   DP_DIAG5[31] := B#16#0;
   DP_DIAG5[32] := B#16#0;
   DP_DIAG5[33] := B#16#0;
   DP_DIAG5[34] := B#16#0;
   DP_DIAG5[35] := B#16#0;
   DP_DIAG5[36] := B#16#0;
   DP_DIAG5[37] := B#16#0;
   DP_DIAG5[38] := B#16#0;
   DP_DIAG5[39] := B#16#0;
   DP_DIAG5[40] := B#16#0;
   DP_DIAG5[41] := B#16#0;
   DP_DIAG5[42] := B#16#0;
   DP_DIAG5[43] := B#16#0;
   DP_DIAG5[44] := B#16#0;
   DP_DIAG5[45] := B#16#0;
   DP_DIAG5[46] := B#16#0;
   DP_DIAG5[47] := B#16#0;
   DP_DIAG5[48] := B#16#0;
   DP_DIAG5[49] := B#16#0;
   DP_DIAG5[50] := B#16#0;
   DP_DIAG5[51] := B#16#0;
   DP_DIAG5[52] := B#16#0;
   DP_DIAG5[53] := B#16#0;
   DP_DIAG5[54] := B#16#0;
   DP_DIAG5[55] := B#16#0;
   DP_DIAG5[56] := B#16#0;
   DP_DIAG5[57] := B#16#0;
   DP_DIAG5[58] := B#16#0;
   DP_DIAG5[59] := B#16#0;
   DP_DIAG5[60] := B#16#0;
   DP_DIAG5[61] := B#16#0;
   DP_DIAG5[62] := B#16#0;
   DP_DIAG5[63] := B#16#0;
   DP_DIAG5[64] := B#16#0;
   DP_DIAG5[65] := B#16#0;
   DP_DIAG5[66] := B#16#0;
   DP_DIAG5[67] := B#16#0;
   DP_DIAG5[68] := B#16#0;
   DP_DIAG5[69] := B#16#0;
   DP_DIAG5[70] := B#16#0;
   DP_DIAG5[71] := B#16#0;
   DP_DIAG5[72] := B#16#0;
   DP_DIAG5[73] := B#16#0;
   DP_DIAG5[74] := B#16#0;
   DP_DIAG5[75] := B#16#0;
   DP_DIAG5[76] := B#16#0;
   DP_DIAG5[77] := B#16#0;
   DP_DIAG5[78] := B#16#0;
   DP_DIAG5[79] := B#16#0;
   DP_DIAG5[80] := B#16#0;
   DP_DIAG5[81] := B#16#0;
   DP_DIAG5[82] := B#16#0;
   DP_DIAG5[83] := B#16#0;
   DP_DIAG5[84] := B#16#0;
   DP_DIAG5[85] := B#16#0;
   DP_DIAG5[86] := B#16#0;
   DP_DIAG5[87] := B#16#0;
   DP_DIAG5[88] := B#16#0;
   DP_DIAG5[89] := B#16#0;
   DP_DIAG5[90] := B#16#0;
   DP_DIAG5[91] := B#16#0;
   DP_DIAG5[92] := B#16#0;
   DP_DIAG5[93] := B#16#0;
   DP_DIAG5[94] := B#16#0;
   DP_DIAG5[95] := B#16#0;
   DP_DIAG5[96] := B#16#0;
   DP_DIAG5[97] := B#16#0;
   DP_DIAG5[98] := B#16#0;
   DP_DIAG5[99] := B#16#0;
   DP_DIAG5[100] := B#16#0;
   DP_DIAG6[1] := B#16#0;
   DP_DIAG6[2] := B#16#0;
   DP_DIAG6[3] := B#16#0;
   DP_DIAG6[4] := B#16#0;
   DP_DIAG6[5] := B#16#0;
   DP_DIAG6[6] := B#16#0;
   DP_DIAG6[7] := B#16#0;
   DP_DIAG6[8] := B#16#0;
   DP_DIAG6[9] := B#16#0;
   DP_DIAG6[10] := B#16#0;
   DP_DIAG6[11] := B#16#0;
   DP_DIAG6[12] := B#16#0;
   DP_DIAG6[13] := B#16#0;
   DP_DIAG6[14] := B#16#0;
   DP_DIAG6[15] := B#16#0;
   DP_DIAG6[16] := B#16#0;
   DP_DIAG6[17] := B#16#0;
   DP_DIAG6[18] := B#16#0;
   DP_DIAG6[19] := B#16#0;
   DP_DIAG6[20] := B#16#0;
   DP_DIAG6[21] := B#16#0;
   DP_DIAG6[22] := B#16#0;
   DP_DIAG6[23] := B#16#0;
   DP_DIAG6[24] := B#16#0;
   DP_DIAG6[25] := B#16#0;
   DP_DIAG6[26] := B#16#0;
   DP_DIAG6[27] := B#16#0;
   DP_DIAG6[28] := B#16#0;
   DP_DIAG6[29] := B#16#0;
   DP_DIAG6[30] := B#16#0;
   DP_DIAG6[31] := B#16#0;
   DP_DIAG6[32] := B#16#0;
   DP_DIAG6[33] := B#16#0;
   DP_DIAG6[34] := B#16#0;
   DP_DIAG6[35] := B#16#0;
   DP_DIAG6[36] := B#16#0;
   DP_DIAG6[37] := B#16#0;
   DP_DIAG6[38] := B#16#0;
   DP_DIAG6[39] := B#16#0;
   DP_DIAG6[40] := B#16#0;
   DP_DIAG6[41] := B#16#0;
   DP_DIAG6[42] := B#16#0;
   DP_DIAG6[43] := B#16#0;
   DP_DIAG6[44] := B#16#0;
   DP_DIAG6[45] := B#16#0;
   DP_DIAG6[46] := B#16#0;
   DP_DIAG6[47] := B#16#0;
   DP_DIAG6[48] := B#16#0;
   DP_DIAG6[49] := B#16#0;
   DP_DIAG6[50] := B#16#0;
   DP_DIAG6[51] := B#16#0;
   DP_DIAG6[52] := B#16#0;
   DP_DIAG6[53] := B#16#0;
   DP_DIAG6[54] := B#16#0;
   DP_DIAG6[55] := B#16#0;
   DP_DIAG6[56] := B#16#0;
   DP_DIAG6[57] := B#16#0;
   DP_DIAG6[58] := B#16#0;
   DP_DIAG6[59] := B#16#0;
   DP_DIAG6[60] := B#16#0;
   DP_DIAG6[61] := B#16#0;
   DP_DIAG6[62] := B#16#0;
   DP_DIAG6[63] := B#16#0;
   DP_DIAG6[64] := B#16#0;
   DP_DIAG6[65] := B#16#0;
   DP_DIAG6[66] := B#16#0;
   DP_DIAG6[67] := B#16#0;
   DP_DIAG6[68] := B#16#0;
   DP_DIAG6[69] := B#16#0;
   DP_DIAG6[70] := B#16#0;
   DP_DIAG6[71] := B#16#0;
   DP_DIAG6[72] := B#16#0;
   DP_DIAG6[73] := B#16#0;
   DP_DIAG6[74] := B#16#0;
   DP_DIAG6[75] := B#16#0;
   DP_DIAG6[76] := B#16#0;
   DP_DIAG6[77] := B#16#0;
   DP_DIAG6[78] := B#16#0;
   DP_DIAG6[79] := B#16#0;
   DP_DIAG6[80] := B#16#0;
   DP_DIAG6[81] := B#16#0;
   DP_DIAG6[82] := B#16#0;
   DP_DIAG6[83] := B#16#0;
   DP_DIAG6[84] := B#16#0;
   DP_DIAG6[85] := B#16#0;
   DP_DIAG6[86] := B#16#0;
   DP_DIAG6[87] := B#16#0;
   DP_DIAG6[88] := B#16#0;
   DP_DIAG6[89] := B#16#0;
   DP_DIAG6[90] := B#16#0;
   DP_DIAG6[91] := B#16#0;
   DP_DIAG6[92] := B#16#0;
   DP_DIAG6[93] := B#16#0;
   DP_DIAG6[94] := B#16#0;
   DP_DIAG6[95] := B#16#0;
   DP_DIAG6[96] := B#16#0;
   DP_DIAG6[97] := B#16#0;
   DP_DIAG6[98] := B#16#0;
   DP_DIAG6[99] := B#16#0;
   DP_DIAG6[100] := B#16#0;
   DP_DIAG7[1] := B#16#0;
   DP_DIAG7[2] := B#16#0;
   DP_DIAG7[3] := B#16#0;
   DP_DIAG7[4] := B#16#0;
   DP_DIAG7[5] := B#16#0;
   DP_DIAG7[6] := B#16#0;
   DP_DIAG7[7] := B#16#0;
   DP_DIAG7[8] := B#16#0;
   DP_DIAG7[9] := B#16#0;
   DP_DIAG7[10] := B#16#0;
   DP_DIAG7[11] := B#16#0;
   DP_DIAG7[12] := B#16#0;
   DP_DIAG7[13] := B#16#0;
   DP_DIAG7[14] := B#16#0;
   DP_DIAG7[15] := B#16#0;
   DP_DIAG7[16] := B#16#0;
   DP_DIAG7[17] := B#16#0;
   DP_DIAG7[18] := B#16#0;
   DP_DIAG7[19] := B#16#0;
   DP_DIAG7[20] := B#16#0;
   DP_DIAG7[21] := B#16#0;
   DP_DIAG7[22] := B#16#0;
   DP_DIAG7[23] := B#16#0;
   DP_DIAG7[24] := B#16#0;
   DP_DIAG7[25] := B#16#0;
   DP_DIAG7[26] := B#16#0;
   DP_DIAG7[27] := B#16#0;
   DP_DIAG7[28] := B#16#0;
   DP_DIAG7[29] := B#16#0;
   DP_DIAG7[30] := B#16#0;
   DP_DIAG7[31] := B#16#0;
   DP_DIAG7[32] := B#16#0;
   DP_DIAG7[33] := B#16#0;
   DP_DIAG7[34] := B#16#0;
   DP_DIAG7[35] := B#16#0;
   DP_DIAG7[36] := B#16#0;
   DP_DIAG7[37] := B#16#0;
   DP_DIAG7[38] := B#16#0;
   DP_DIAG7[39] := B#16#0;
   DP_DIAG7[40] := B#16#0;
   DP_DIAG7[41] := B#16#0;
   DP_DIAG7[42] := B#16#0;
   DP_DIAG7[43] := B#16#0;
   DP_DIAG7[44] := B#16#0;
   DP_DIAG7[45] := B#16#0;
   DP_DIAG7[46] := B#16#0;
   DP_DIAG7[47] := B#16#0;
   DP_DIAG7[48] := B#16#0;
   DP_DIAG7[49] := B#16#0;
   DP_DIAG7[50] := B#16#0;
   DP_DIAG7[51] := B#16#0;
   DP_DIAG7[52] := B#16#0;
   DP_DIAG7[53] := B#16#0;
   DP_DIAG7[54] := B#16#0;
   DP_DIAG7[55] := B#16#0;
   DP_DIAG7[56] := B#16#0;
   DP_DIAG7[57] := B#16#0;
   DP_DIAG7[58] := B#16#0;
   DP_DIAG7[59] := B#16#0;
   DP_DIAG7[60] := B#16#0;
   DP_DIAG7[61] := B#16#0;
   DP_DIAG7[62] := B#16#0;
   DP_DIAG7[63] := B#16#0;
   DP_DIAG7[64] := B#16#0;
   DP_DIAG7[65] := B#16#0;
   DP_DIAG7[66] := B#16#0;
   DP_DIAG7[67] := B#16#0;
   DP_DIAG7[68] := B#16#0;
   DP_DIAG7[69] := B#16#0;
   DP_DIAG7[70] := B#16#0;
   DP_DIAG7[71] := B#16#0;
   DP_DIAG7[72] := B#16#0;
   DP_DIAG7[73] := B#16#0;
   DP_DIAG7[74] := B#16#0;
   DP_DIAG7[75] := B#16#0;
   DP_DIAG7[76] := B#16#0;
   DP_DIAG7[77] := B#16#0;
   DP_DIAG7[78] := B#16#0;
   DP_DIAG7[79] := B#16#0;
   DP_DIAG7[80] := B#16#0;
   DP_DIAG7[81] := B#16#0;
   DP_DIAG7[82] := B#16#0;
   DP_DIAG7[83] := B#16#0;
   DP_DIAG7[84] := B#16#0;
   DP_DIAG7[85] := B#16#0;
   DP_DIAG7[86] := B#16#0;
   DP_DIAG7[87] := B#16#0;
   DP_DIAG7[88] := B#16#0;
   DP_DIAG7[89] := B#16#0;
   DP_DIAG7[90] := B#16#0;
   DP_DIAG7[91] := B#16#0;
   DP_DIAG7[92] := B#16#0;
   DP_DIAG7[93] := B#16#0;
   DP_DIAG7[94] := B#16#0;
   DP_DIAG7[95] := B#16#0;
   DP_DIAG7[96] := B#16#0;
   DP_DIAG7[97] := B#16#0;
   DP_DIAG7[98] := B#16#0;
   DP_DIAG7[99] := B#16#0;
   DP_DIAG7[100] := B#16#0;
   DP_DIAG8[1] := B#16#0;
   DP_DIAG8[2] := B#16#0;
   DP_DIAG8[3] := B#16#0;
   DP_DIAG8[4] := B#16#0;
   DP_DIAG8[5] := B#16#0;
   DP_DIAG8[6] := B#16#0;
   DP_DIAG8[7] := B#16#0;
   DP_DIAG8[8] := B#16#0;
   DP_DIAG8[9] := B#16#0;
   DP_DIAG8[10] := B#16#0;
   DP_DIAG8[11] := B#16#0;
   DP_DIAG8[12] := B#16#0;
   DP_DIAG8[13] := B#16#0;
   DP_DIAG8[14] := B#16#0;
   DP_DIAG8[15] := B#16#0;
   DP_DIAG8[16] := B#16#0;
   DP_DIAG8[17] := B#16#0;
   DP_DIAG8[18] := B#16#0;
   DP_DIAG8[19] := B#16#0;
   DP_DIAG8[20] := B#16#0;
   DP_DIAG8[21] := B#16#0;
   DP_DIAG8[22] := B#16#0;
   DP_DIAG8[23] := B#16#0;
   DP_DIAG8[24] := B#16#0;
   DP_DIAG8[25] := B#16#0;
   DP_DIAG8[26] := B#16#0;
   DP_DIAG8[27] := B#16#0;
   DP_DIAG8[28] := B#16#0;
   DP_DIAG8[29] := B#16#0;
   DP_DIAG8[30] := B#16#0;
   DP_DIAG8[31] := B#16#0;
   DP_DIAG8[32] := B#16#0;
   DP_DIAG8[33] := B#16#0;
   DP_DIAG8[34] := B#16#0;
   DP_DIAG8[35] := B#16#0;
   DP_DIAG8[36] := B#16#0;
   DP_DIAG8[37] := B#16#0;
   DP_DIAG8[38] := B#16#0;
   DP_DIAG8[39] := B#16#0;
   DP_DIAG8[40] := B#16#0;
   DP_DIAG8[41] := B#16#0;
   DP_DIAG8[42] := B#16#0;
   DP_DIAG8[43] := B#16#0;
   DP_DIAG8[44] := B#16#0;
   DP_DIAG8[45] := B#16#0;
   DP_DIAG8[46] := B#16#0;
   DP_DIAG8[47] := B#16#0;
   DP_DIAG8[48] := B#16#0;
   DP_DIAG8[49] := B#16#0;
   DP_DIAG8[50] := B#16#0;
   DP_DIAG8[51] := B#16#0;
   DP_DIAG8[52] := B#16#0;
   DP_DIAG8[53] := B#16#0;
   DP_DIAG8[54] := B#16#0;
   DP_DIAG8[55] := B#16#0;
   DP_DIAG8[56] := B#16#0;
   DP_DIAG8[57] := B#16#0;
   DP_DIAG8[58] := B#16#0;
   DP_DIAG8[59] := B#16#0;
   DP_DIAG8[60] := B#16#0;
   DP_DIAG8[61] := B#16#0;
   DP_DIAG8[62] := B#16#0;
   DP_DIAG8[63] := B#16#0;
   DP_DIAG8[64] := B#16#0;
   DP_DIAG8[65] := B#16#0;
   DP_DIAG8[66] := B#16#0;
   DP_DIAG8[67] := B#16#0;
   DP_DIAG8[68] := B#16#0;
   DP_DIAG8[69] := B#16#0;
   DP_DIAG8[70] := B#16#0;
   DP_DIAG8[71] := B#16#0;
   DP_DIAG8[72] := B#16#0;
   DP_DIAG8[73] := B#16#0;
   DP_DIAG8[74] := B#16#0;
   DP_DIAG8[75] := B#16#0;
   DP_DIAG8[76] := B#16#0;
   DP_DIAG8[77] := B#16#0;
   DP_DIAG8[78] := B#16#0;
   DP_DIAG8[79] := B#16#0;
   DP_DIAG8[80] := B#16#0;
   DP_DIAG8[81] := B#16#0;
   DP_DIAG8[82] := B#16#0;
   DP_DIAG8[83] := B#16#0;
   DP_DIAG8[84] := B#16#0;
   DP_DIAG8[85] := B#16#0;
   DP_DIAG8[86] := B#16#0;
   DP_DIAG8[87] := B#16#0;
   DP_DIAG8[88] := B#16#0;
   DP_DIAG8[89] := B#16#0;
   DP_DIAG8[90] := B#16#0;
   DP_DIAG8[91] := B#16#0;
   DP_DIAG8[92] := B#16#0;
   DP_DIAG8[93] := B#16#0;
   DP_DIAG8[94] := B#16#0;
   DP_DIAG8[95] := B#16#0;
   DP_DIAG8[96] := B#16#0;
   DP_DIAG8[97] := B#16#0;
   DP_DIAG8[98] := B#16#0;
   DP_DIAG8[99] := B#16#0;
   DP_DIAG8[100] := B#16#0;
   DP_DIAG9[1] := B#16#0;
   DP_DIAG9[2] := B#16#0;
   DP_DIAG9[3] := B#16#0;
   DP_DIAG9[4] := B#16#0;
   DP_DIAG9[5] := B#16#0;
   DP_DIAG9[6] := B#16#0;
   DP_DIAG9[7] := B#16#0;
   DP_DIAG9[8] := B#16#0;
   DP_DIAG9[9] := B#16#0;
   DP_DIAG9[10] := B#16#0;
   DP_DIAG9[11] := B#16#0;
   DP_DIAG9[12] := B#16#0;
   DP_DIAG9[13] := B#16#0;
   DP_DIAG9[14] := B#16#0;
   DP_DIAG9[15] := B#16#0;
   DP_DIAG9[16] := B#16#0;
   DP_DIAG9[17] := B#16#0;
   DP_DIAG9[18] := B#16#0;
   DP_DIAG9[19] := B#16#0;
   DP_DIAG9[20] := B#16#0;
   DP_DIAG9[21] := B#16#0;
   DP_DIAG9[22] := B#16#0;
   DP_DIAG9[23] := B#16#0;
   DP_DIAG9[24] := B#16#0;
   DP_DIAG9[25] := B#16#0;
   DP_DIAG9[26] := B#16#0;
   DP_DIAG9[27] := B#16#0;
   DP_DIAG9[28] := B#16#0;
   DP_DIAG9[29] := B#16#0;
   DP_DIAG9[30] := B#16#0;
   DP_DIAG9[31] := B#16#0;
   DP_DIAG9[32] := B#16#0;
   DP_DIAG9[33] := B#16#0;
   DP_DIAG9[34] := B#16#0;
   DP_DIAG9[35] := B#16#0;
   DP_DIAG9[36] := B#16#0;
   DP_DIAG9[37] := B#16#0;
   DP_DIAG9[38] := B#16#0;
   DP_DIAG9[39] := B#16#0;
   DP_DIAG9[40] := B#16#0;
   DP_DIAG9[41] := B#16#0;
   DP_DIAG9[42] := B#16#0;
   DP_DIAG9[43] := B#16#0;
   DP_DIAG9[44] := B#16#0;
   DP_DIAG9[45] := B#16#0;
   DP_DIAG9[46] := B#16#0;
   DP_DIAG9[47] := B#16#0;
   DP_DIAG9[48] := B#16#0;
   DP_DIAG9[49] := B#16#0;
   DP_DIAG9[50] := B#16#0;
   DP_DIAG9[51] := B#16#0;
   DP_DIAG9[52] := B#16#0;
   DP_DIAG9[53] := B#16#0;
   DP_DIAG9[54] := B#16#0;
   DP_DIAG9[55] := B#16#0;
   DP_DIAG9[56] := B#16#0;
   DP_DIAG9[57] := B#16#0;
   DP_DIAG9[58] := B#16#0;
   DP_DIAG9[59] := B#16#0;
   DP_DIAG9[60] := B#16#0;
   DP_DIAG9[61] := B#16#0;
   DP_DIAG9[62] := B#16#0;
   DP_DIAG9[63] := B#16#0;
   DP_DIAG9[64] := B#16#0;
   DP_DIAG9[65] := B#16#0;
   DP_DIAG9[66] := B#16#0;
   DP_DIAG9[67] := B#16#0;
   DP_DIAG9[68] := B#16#0;
   DP_DIAG9[69] := B#16#0;
   DP_DIAG9[70] := B#16#0;
   DP_DIAG9[71] := B#16#0;
   DP_DIAG9[72] := B#16#0;
   DP_DIAG9[73] := B#16#0;
   DP_DIAG9[74] := B#16#0;
   DP_DIAG9[75] := B#16#0;
   DP_DIAG9[76] := B#16#0;
   DP_DIAG9[77] := B#16#0;
   DP_DIAG9[78] := B#16#0;
   DP_DIAG9[79] := B#16#0;
   DP_DIAG9[80] := B#16#0;
   DP_DIAG9[81] := B#16#0;
   DP_DIAG9[82] := B#16#0;
   DP_DIAG9[83] := B#16#0;
   DP_DIAG9[84] := B#16#0;
   DP_DIAG9[85] := B#16#0;
   DP_DIAG9[86] := B#16#0;
   DP_DIAG9[87] := B#16#0;
   DP_DIAG9[88] := B#16#0;
   DP_DIAG9[89] := B#16#0;
   DP_DIAG9[90] := B#16#0;
   DP_DIAG9[91] := B#16#0;
   DP_DIAG9[92] := B#16#0;
   DP_DIAG9[93] := B#16#0;
   DP_DIAG9[94] := B#16#0;
   DP_DIAG9[95] := B#16#0;
   DP_DIAG9[96] := B#16#0;
   DP_DIAG9[97] := B#16#0;
   DP_DIAG9[98] := B#16#0;
   DP_DIAG9[99] := B#16#0;
   DP_DIAG9[100] := B#16#0;
   DP_DIAG10[1] := B#16#0;
   DP_DIAG10[2] := B#16#0;
   DP_DIAG10[3] := B#16#0;
   DP_DIAG10[4] := B#16#0;
   DP_DIAG10[5] := B#16#0;
   DP_DIAG10[6] := B#16#0;
   DP_DIAG10[7] := B#16#0;
   DP_DIAG10[8] := B#16#0;
   DP_DIAG10[9] := B#16#0;
   DP_DIAG10[10] := B#16#0;
   DP_DIAG10[11] := B#16#0;
   DP_DIAG10[12] := B#16#0;
   DP_DIAG10[13] := B#16#0;
   DP_DIAG10[14] := B#16#0;
   DP_DIAG10[15] := B#16#0;
   DP_DIAG10[16] := B#16#0;
   DP_DIAG10[17] := B#16#0;
   DP_DIAG10[18] := B#16#0;
   DP_DIAG10[19] := B#16#0;
   DP_DIAG10[20] := B#16#0;
   DP_DIAG10[21] := B#16#0;
   DP_DIAG10[22] := B#16#0;
   DP_DIAG10[23] := B#16#0;
   DP_DIAG10[24] := B#16#0;
   DP_DIAG10[25] := B#16#0;
   DP_DIAG10[26] := B#16#0;
   DP_DIAG10[27] := B#16#0;
   DP_DIAG10[28] := B#16#0;
   DP_DIAG10[29] := B#16#0;
   DP_DIAG10[30] := B#16#0;
   DP_DIAG10[31] := B#16#0;
   DP_DIAG10[32] := B#16#0;
   DP_DIAG10[33] := B#16#0;
   DP_DIAG10[34] := B#16#0;
   DP_DIAG10[35] := B#16#0;
   DP_DIAG10[36] := B#16#0;
   DP_DIAG10[37] := B#16#0;
   DP_DIAG10[38] := B#16#0;
   DP_DIAG10[39] := B#16#0;
   DP_DIAG10[40] := B#16#0;
   DP_DIAG10[41] := B#16#0;
   DP_DIAG10[42] := B#16#0;
   DP_DIAG10[43] := B#16#0;
   DP_DIAG10[44] := B#16#0;
   DP_DIAG10[45] := B#16#0;
   DP_DIAG10[46] := B#16#0;
   DP_DIAG10[47] := B#16#0;
   DP_DIAG10[48] := B#16#0;
   DP_DIAG10[49] := B#16#0;
   DP_DIAG10[50] := B#16#0;
   DP_DIAG10[51] := B#16#0;
   DP_DIAG10[52] := B#16#0;
   DP_DIAG10[53] := B#16#0;
   DP_DIAG10[54] := B#16#0;
   DP_DIAG10[55] := B#16#0;
   DP_DIAG10[56] := B#16#0;
   DP_DIAG10[57] := B#16#0;
   DP_DIAG10[58] := B#16#0;
   DP_DIAG10[59] := B#16#0;
   DP_DIAG10[60] := B#16#0;
   DP_DIAG10[61] := B#16#0;
   DP_DIAG10[62] := B#16#0;
   DP_DIAG10[63] := B#16#0;
   DP_DIAG10[64] := B#16#0;
   DP_DIAG10[65] := B#16#0;
   DP_DIAG10[66] := B#16#0;
   DP_DIAG10[67] := B#16#0;
   DP_DIAG10[68] := B#16#0;
   DP_DIAG10[69] := B#16#0;
   DP_DIAG10[70] := B#16#0;
   DP_DIAG10[71] := B#16#0;
   DP_DIAG10[72] := B#16#0;
   DP_DIAG10[73] := B#16#0;
   DP_DIAG10[74] := B#16#0;
   DP_DIAG10[75] := B#16#0;
   DP_DIAG10[76] := B#16#0;
   DP_DIAG10[77] := B#16#0;
   DP_DIAG10[78] := B#16#0;
   DP_DIAG10[79] := B#16#0;
   DP_DIAG10[80] := B#16#0;
   DP_DIAG10[81] := B#16#0;
   DP_DIAG10[82] := B#16#0;
   DP_DIAG10[83] := B#16#0;
   DP_DIAG10[84] := B#16#0;
   DP_DIAG10[85] := B#16#0;
   DP_DIAG10[86] := B#16#0;
   DP_DIAG10[87] := B#16#0;
   DP_DIAG10[88] := B#16#0;
   DP_DIAG10[89] := B#16#0;
   DP_DIAG10[90] := B#16#0;
   DP_DIAG10[91] := B#16#0;
   DP_DIAG10[92] := B#16#0;
   DP_DIAG10[93] := B#16#0;
   DP_DIAG10[94] := B#16#0;
   DP_DIAG10[95] := B#16#0;
   DP_DIAG10[96] := B#16#0;
   DP_DIAG10[97] := B#16#0;
   DP_DIAG10[98] := B#16#0;
   DP_DIAG10[99] := B#16#0;
   DP_DIAG10[100] := B#16#0;
END_DATA_BLOCK

FUNCTION_BLOCK FB 402
TITLE =Operation Mode Select Program
AUTHOR : HMC
FAMILY : Mode
NAME : Mode
VERSION : 1.0


VAR_INPUT
  SSD_Manual : BOOL ;
  SSD_Auto : BOOL ;
  PB_Ready : BOOL ;
  PB_Auto_Run : BOOL ;
  PB_Remote_Ready : BOOL ;
  PB_Remote_Auto_Run : BOOL ;
  PB_Lamp_CHK : BOOL ;
  M_Air_Error : BOOL ;
  M_Water_Error : BOOL ;
  M_Total_Error : BOOL ;
  M_EStop : BOOL ;
  EXT_Ready : BOOL ;
  EXT_Auto : BOOL ;
  T_SemiAuto : TIME ;
  M_FLICK : BOOL ;
END_VAR
VAR_OUTPUT
  M_Ready_On : BOOL ;
  M_Auto_Mode : BOOL ;
  M_SemiAuto_Mode : BOOL ;
  M_Manual_Mode : BOOL ;
  M_Auto_Run : BOOL ;
  LP_Ready_On : BOOL ;
  LP_Auto_Run : BOOL ;
END_VAR
VAR
  AUTO_MODE_DELAY : SFB 4;
  SEMI_AUTO_DELAY : SFB 4;
  MANUAL_DELAY : SFB 4;
END_VAR
BEGIN
NETWORK
TITLE =Auto Mode Select Program
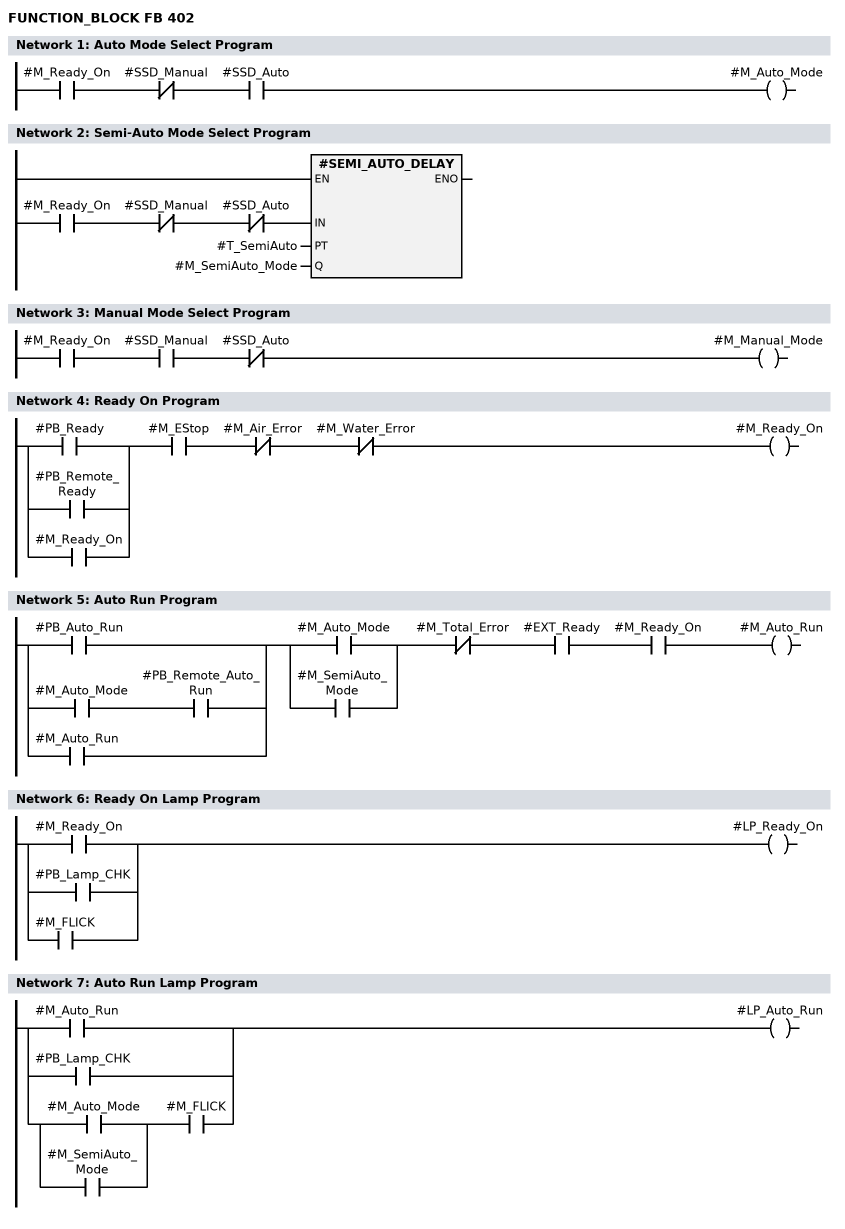

      A     #M_Ready_On;
      AN    #SSD_Manual;
      A     #SSD_Auto;
      =     #M_Auto_Mode;
NETWORK
TITLE =Semi-Auto Mode Select Program

      A     #M_Ready_On;
      AN    #SSD_Manual;
      AN    #SSD_Auto;
      =     L      0.0;
      BLD   103;
      CALL #SEMI_AUTO_DELAY (
           IN                       := L      0.0,
           PT                       := #T_SemiAuto,
           Q                        := #M_SemiAuto_Mode);

      NOP   0;
NETWORK
TITLE =Manual Mode Select Program

      A     #M_Ready_On;
      A     #SSD_Manual;
      AN    #SSD_Auto;
      =     #M_Manual_Mode;
NETWORK
TITLE =Ready On Program

      A(    ;
      O     #PB_Ready;
      O     #PB_Remote_Ready;
      O     #M_Ready_On;
      )     ;
      A     #M_EStop;
      AN    #M_Air_Error;
      AN    #M_Water_Error;
      =     #M_Ready_On;
NETWORK
TITLE =Auto Run Program

      A(    ;
      O     #PB_Auto_Run;
      O     ;
      A     #M_Auto_Mode;
      A     #PB_Remote_Auto_Run;
      O     #M_Auto_Run;
      )     ;
      A(    ;
      O     #M_Auto_Mode;
      O     #M_SemiAuto_Mode;
      )     ;
      AN    #M_Total_Error;
      A     #EXT_Ready;
      A     #M_Ready_On;
      =     #M_Auto_Run;
NETWORK
TITLE =Ready On Lamp Program

      O     #M_Ready_On;
      O     #PB_Lamp_CHK;
      O     #M_FLICK;
      =     #LP_Ready_On;
NETWORK
TITLE =Auto Run Lamp Program

      O     #M_Auto_Run;
      O     #PB_Lamp_CHK;
      O     ;
      A(    ;
      O     #M_Auto_Mode;
      O     #M_SemiAuto_Mode;
      )     ;
      A     #M_FLICK;
      =     #LP_Auto_Run;
END_FUNCTION_BLOCK

FUNCTION_BLOCK FB 424
TITLE =Sensor Error,Lamp Variables Program
AUTHOR : HMC
FAMILY : Common
NAME : Common
VERSION : 1.0


VAR_INPUT
  Enable_Aux : BOOL ;
  Adv_Amount : INT ;
  Ret_Amount : INT ;
  LS_Adv1 : BOOL ;
  LS_Ret1 : BOOL ;
  LS_Adv2 : BOOL ;
  LS_Ret2 : BOOL ;
  LS_Adv3 : BOOL ;
  LS_Ret3 : BOOL ;
  LS_Adv4 : BOOL ;
  LS_Ret4 : BOOL ;
  SOL_Adv : BOOL ;
  SOL_Ret : BOOL ;
  M_Ready : BOOL ;
  T_CHK1 : TIME ;
  T_CHK2 : TIME ;
  PB_Lamp_CHK : BOOL ;
  PB_Error_Rst : BOOL ;
  M_FLICK : BOOL ;
END_VAR
VAR_OUTPUT
  M_Adv_Err : BOOL ;
  M_Ret_Err : BOOL ;
  LP_Adv : BOOL ;
  LP_Ret : BOOL ;
  Visu_Adv : WORD ;
  Visu_Ret : WORD ;
END_VAR
VAR
  Error_T1 : SFB 4;
  Error_T2 : SFB 4;
  CHK_Aux1 : BOOL ;
  CHK_Aux2 : BOOL ;
  Error_T1_DN : BOOL ;
  Error_T2_DN : BOOL ;
  Adv_Memo : BOOL ;
  Visu_Adv_Arr : ARRAY  [0 .. 15 ] OF BOOL ;
  Visu_Ret_Arr : ARRAY  [0 .. 15 ] OF BOOL ;
  BLK_Move_Ret : INT ;
  Enable : BOOL ;
  Adv_End : BOOL ;
  Ret_End : BOOL ;
END_VAR
BEGIN
NETWORK
TITLE =
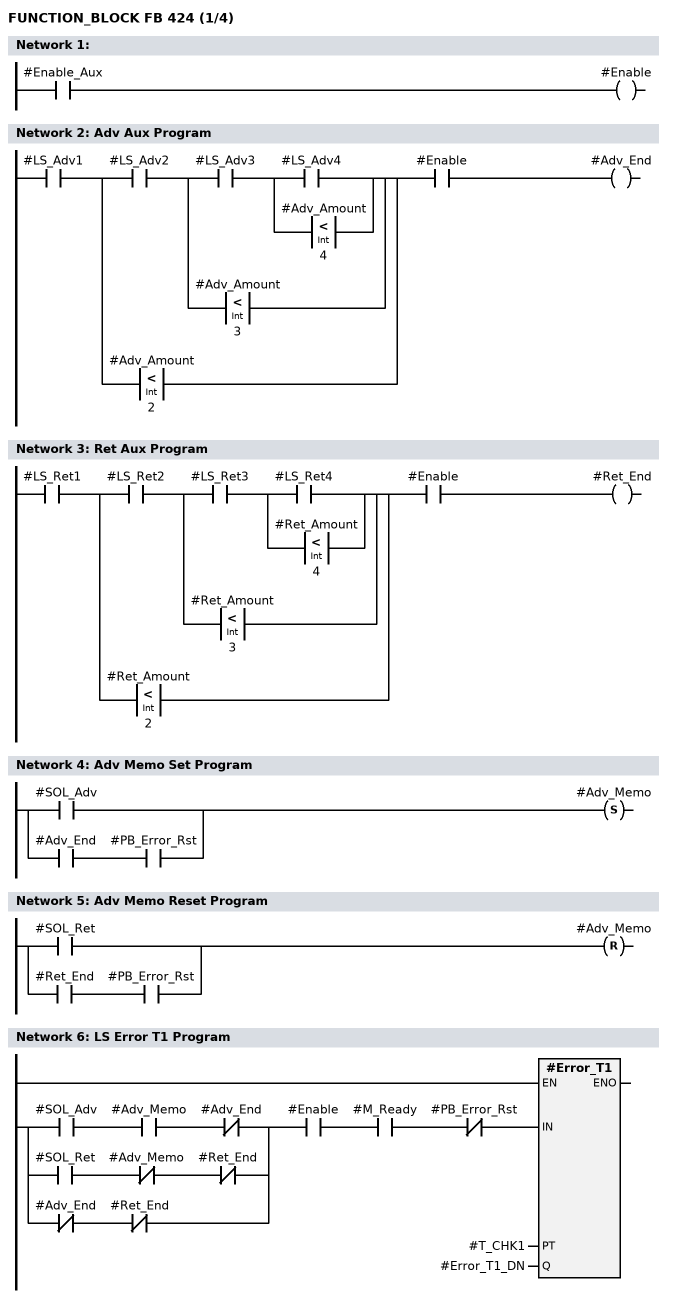

      A     #Enable_Aux;
      =     #Enable;
NETWORK
TITLE =Adv Aux Program

      A     #LS_Adv1;
      A(    ;
      A     #LS_Adv2;
      A(    ;
      A     #LS_Adv3;
      A(    ;
      O     #LS_Adv4;
      O(    ;
      L     #Adv_Amount;
      L     4;
      <I    ;
      )     ;
      )     ;
      O(    ;
      L     #Adv_Amount;
      L     3;
      <I    ;
      )     ;
      )     ;
      O(    ;
      L     #Adv_Amount;
      L     2;
      <I    ;
      )     ;
      )     ;
      A     #Enable;
      =     #Adv_End;
NETWORK
TITLE =Ret Aux Program

      A     #LS_Ret1;
      A(    ;
      A     #LS_Ret2;
      A(    ;
      A     #LS_Ret3;
      A(    ;
      O     #LS_Ret4;
      O(    ;
      L     #Ret_Amount;
      L     4;
      <I    ;
      )     ;
      )     ;
      O(    ;
      L     #Ret_Amount;
      L     3;
      <I    ;
      )     ;
      )     ;
      O(    ;
      L     #Ret_Amount;
      L     2;
      <I    ;
      )     ;
      )     ;
      A     #Enable;
      =     #Ret_End;
NETWORK
TITLE =Adv Memo Set Program

      O     #SOL_Adv;
      O     ;
      A     #Adv_End;
      A     #PB_Error_Rst;
      S     #Adv_Memo;
NETWORK
TITLE =Adv Memo Reset Program

      O     #SOL_Ret;
      O     ;
      A     #Ret_End;
      A     #PB_Error_Rst;
      R     #Adv_Memo;
NETWORK
TITLE =LS Error T1 Program

      A(    ;
      A     #SOL_Adv;
      A     #Adv_Memo;
      AN    #Adv_End;
      O     ;
      A     #SOL_Ret;
      AN    #Adv_Memo;
      AN    #Ret_End;
      O     ;
      AN    #Adv_End;
      AN    #Ret_End;
      )     ;
      A     #Enable;
      A     #M_Ready;
      AN    #PB_Error_Rst;
      =     L      0.0;
      BLD   103;
      CALL #Error_T1 (
           IN                       := L      0.0,
           PT                       := #T_CHK1,
           Q                        := #Error_T1_DN);

      NOP   0;
NETWORK
TITLE =Check Aux1 Program
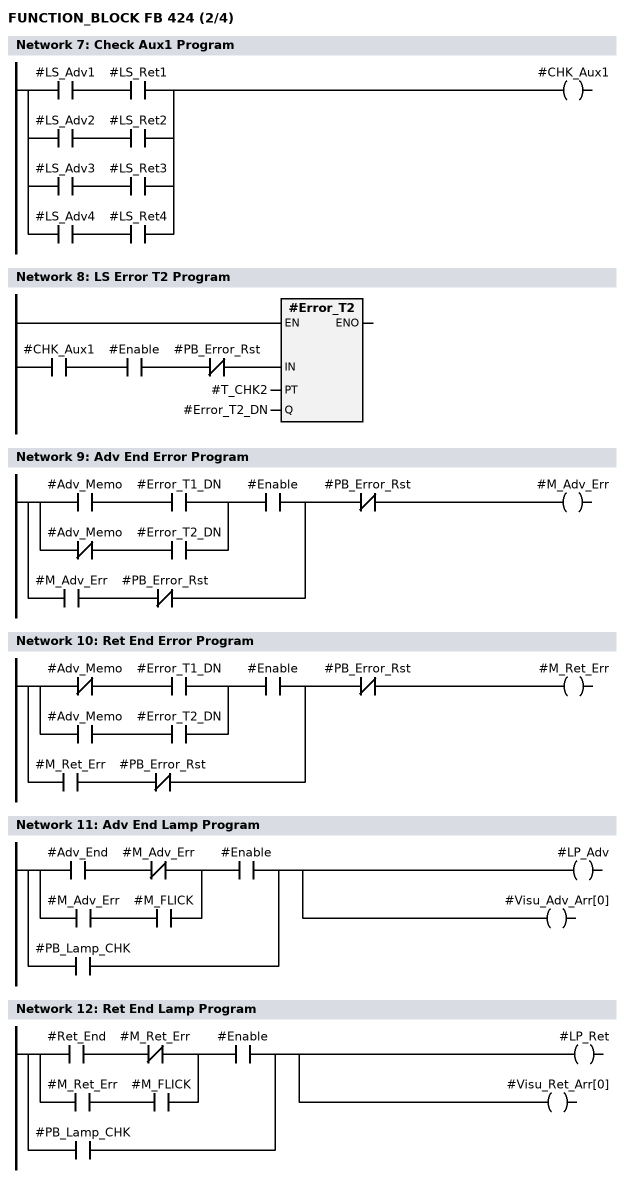

      A     #LS_Adv1;
      A     #LS_Ret1;
      O     ;
      A     #LS_Adv2;
      A     #LS_Ret2;
      O     ;
      A     #LS_Adv3;
      A     #LS_Ret3;
      O     ;
      A     #LS_Adv4;
      A     #LS_Ret4;
      =     #CHK_Aux1;
NETWORK
TITLE =LS Error T2 Program

      A     #CHK_Aux1;
      A     #Enable;
      AN    #PB_Error_Rst;
      =     L      0.0;
      BLD   103;
      CALL #Error_T2 (
           IN                       := L      0.0,
           PT                       := #T_CHK2,
           Q                        := #Error_T2_DN);

      NOP   0;
NETWORK
TITLE =Adv End Error Program

      A(    ;
      A(    ;
      A     #Adv_Memo;
      A     #Error_T1_DN;
      O     ;
      AN    #Adv_Memo;
      A     #Error_T2_DN;
      )     ;
      A     #Enable;
      O     ;
      A     #M_Adv_Err;
      AN    #PB_Error_Rst;
      )     ;
      AN    #PB_Error_Rst;
      =     #M_Adv_Err;
NETWORK
TITLE =Ret End Error Program

      A(    ;
      A(    ;
      AN    #Adv_Memo;
      A     #Error_T1_DN;
      O     ;
      A     #Adv_Memo;
      A     #Error_T2_DN;
      )     ;
      A     #Enable;
      O     ;
      A     #M_Ret_Err;
      AN    #PB_Error_Rst;
      )     ;
      AN    #PB_Error_Rst;
      =     #M_Ret_Err;
NETWORK
TITLE =Adv End Lamp Program

      A(    ;
      A     #Adv_End;
      AN    #M_Adv_Err;
      O     ;
      A     #M_Adv_Err;
      A     #M_FLICK;
      )     ;
      A     #Enable;
      O     #PB_Lamp_CHK;
      =     #LP_Adv;
      =     #Visu_Adv_Arr[0];
NETWORK
TITLE =Ret End Lamp Program

      A(    ;
      A     #Ret_End;
      AN    #M_Ret_Err;
      O     ;
      A     #M_Ret_Err;
      A     #M_FLICK;
      )     ;
      A     #Enable;
      O     #PB_Lamp_CHK;
      =     #LP_Ret;
      =     #Visu_Ret_Arr[0];
NETWORK
TITLE =Adv LS_1 Lamp Program
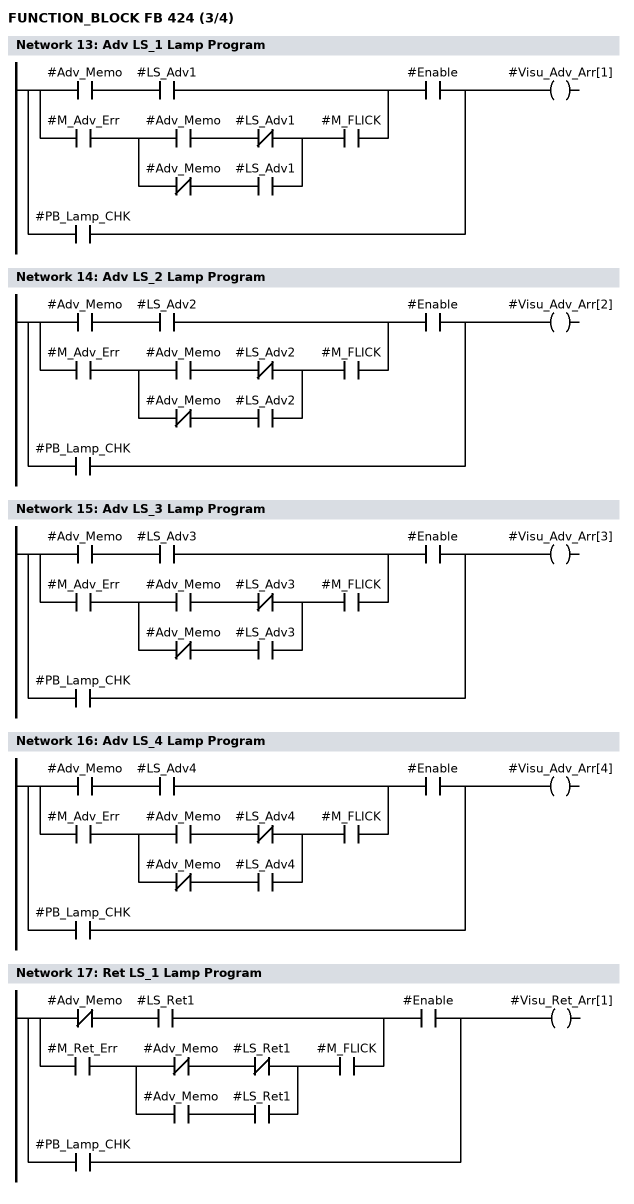

      A(    ;
      A     #Adv_Memo;
      A     #LS_Adv1;
      O     ;
      A     #M_Adv_Err;
      A(    ;
      A     #Adv_Memo;
      AN    #LS_Adv1;
      O     ;
      AN    #Adv_Memo;
      A     #LS_Adv1;
      )     ;
      A     #M_FLICK;
      )     ;
      A     #Enable;
      O     #PB_Lamp_CHK;
      =     #Visu_Adv_Arr[1];
NETWORK
TITLE =Adv LS_2 Lamp Program
//
//
      A(    ;
      A     #Adv_Memo;
      A     #LS_Adv2;
      O     ;
      A     #M_Adv_Err;
      A(    ;
      A     #Adv_Memo;
      AN    #LS_Adv2;
      O     ;
      AN    #Adv_Memo;
      A     #LS_Adv2;
      )     ;
      A     #M_FLICK;
      )     ;
      A     #Enable;
      O     #PB_Lamp_CHK;
      =     #Visu_Adv_Arr[2];
NETWORK
TITLE =Adv LS_3 Lamp Program
//
//
      A(    ;
      A     #Adv_Memo;
      A     #LS_Adv3;
      O     ;
      A     #M_Adv_Err;
      A(    ;
      A     #Adv_Memo;
      AN    #LS_Adv3;
      O     ;
      AN    #Adv_Memo;
      A     #LS_Adv3;
      )     ;
      A     #M_FLICK;
      )     ;
      A     #Enable;
      O     #PB_Lamp_CHK;
      =     #Visu_Adv_Arr[3];
NETWORK
TITLE =Adv LS_4 Lamp Program
//
//
      A(    ;
      A     #Adv_Memo;
      A     #LS_Adv4;
      O     ;
      A     #M_Adv_Err;
      A(    ;
      A     #Adv_Memo;
      AN    #LS_Adv4;
      O     ;
      AN    #Adv_Memo;
      A     #LS_Adv4;
      )     ;
      A     #M_FLICK;
      )     ;
      A     #Enable;
      O     #PB_Lamp_CHK;
      =     #Visu_Adv_Arr[4];
NETWORK
TITLE =Ret LS_1 Lamp Program
//
//
      A(    ;
      AN    #Adv_Memo;
      A     #LS_Ret1;
      O     ;
      A     #M_Ret_Err;
      A(    ;
      AN    #Adv_Memo;
      AN    #LS_Ret1;
      O     ;
      A     #Adv_Memo;
      A     #LS_Ret1;
      )     ;
      A     #M_FLICK;
      )     ;
      A     #Enable;
      O     #PB_Lamp_CHK;
      =     #Visu_Ret_Arr[1];
NETWORK
TITLE =Ret LS_2 Lamp Program
//
//
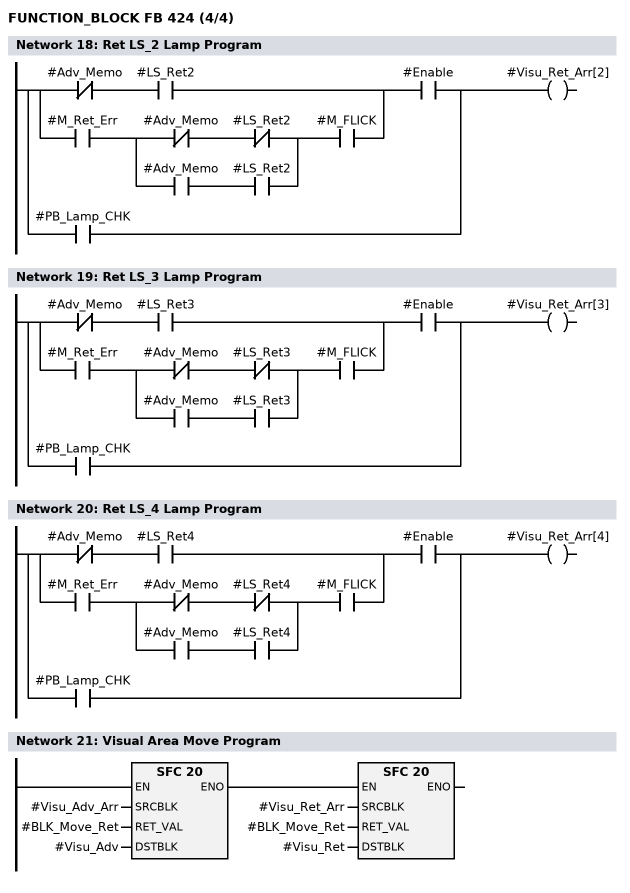
      A(    ;
      AN    #Adv_Memo;
      A     #LS_Ret2;
      O     ;
      A     #M_Ret_Err;
      A(    ;
      AN    #Adv_Memo;
      AN    #LS_Ret2;
      O     ;
      A     #Adv_Memo;
      A     #LS_Ret2;
      )     ;
      A     #M_FLICK;
      )     ;
      A     #Enable;
      O     #PB_Lamp_CHK;
      =     #Visu_Ret_Arr[2];
NETWORK
TITLE =Ret LS_3 Lamp Program
//
//
      A(    ;
      AN    #Adv_Memo;
      A     #LS_Ret3;
      O     ;
      A     #M_Ret_Err;
      A(    ;
      AN    #Adv_Memo;
      AN    #LS_Ret3;
      O     ;
      A     #Adv_Memo;
      A     #LS_Ret3;
      )     ;
      A     #M_FLICK;
      )     ;
      A     #Enable;
      O     #PB_Lamp_CHK;
      =     #Visu_Ret_Arr[3];
NETWORK
TITLE =Ret LS_4 Lamp Program
//
//
      A(    ;
      AN    #Adv_Memo;
      A     #LS_Ret4;
      O     ;
      A     #M_Ret_Err;
      A(    ;
      AN    #Adv_Memo;
      AN    #LS_Ret4;
      O     ;
      A     #Adv_Memo;
      A     #LS_Ret4;
      )     ;
      A     #M_FLICK;
      )     ;
      A     #Enable;
      O     #PB_Lamp_CHK;
      =     #Visu_Ret_Arr[4];
NETWORK
TITLE =Visual Area Move Program

      A(    ;
      CALL SFC   20 (
           SRCBLK                   := #Visu_Adv_Arr,
           RET_VAL                  := #BLK_Move_Ret,
           DSTBLK                   := #Visu_Adv);
      A     BR;
      )     ;
      JNB   _001;
      CALL SFC   20 (
           SRCBLK                   := #Visu_Ret_Arr,
           RET_VAL                  := #BLK_Move_Ret,
           DSTBLK                   := #Visu_Ret);
_001: NOP   0;
END_FUNCTION_BLOCK

FUNCTION_BLOCK FB 426
TITLE =Sensor Error,Lamp Variables Program
AUTHOR : HMC
FAMILY : Common
NAME : Common
VERSION : 1.0


VAR_INPUT
  Enable_Aux : BOOL ;
  Adv_Amount : INT ;
  Ret_Amount : INT ;
  LS_Adv1 : BOOL ;
  LS_Ret1 : BOOL ;
  LS_Adv2 : BOOL ;
  LS_Ret2 : BOOL ;
  LS_Adv3 : BOOL ;
  LS_Ret3 : BOOL ;
  LS_Adv4 : BOOL ;
  LS_Ret4 : BOOL ;
  LS_Adv5 : BOOL ;
  LS_Ret5 : BOOL ;
  LS_Adv6 : BOOL ;
  LS_Ret6 : BOOL ;
  LS_Adv7 : BOOL ;
  LS_Ret7 : BOOL ;
  LS_Adv8 : BOOL ;
  LS_Ret8 : BOOL ;
  SOL_Adv : BOOL ;
  SOL_Ret : BOOL ;
  M_Ready : BOOL ;
  T_CHK1 : TIME ;
  T_CHK2 : TIME ;
  PB_Lamp_CHK : BOOL ;
  PB_Error_Rst : BOOL ;
  M_FLICK : BOOL ;
END_VAR
VAR_OUTPUT
  M_Adv_Err : BOOL ;
  M_Ret_Err : BOOL ;
  LP_Adv : BOOL ;
  LP_Ret : BOOL ;
  Visu_Adv : WORD ;
  Visu_Ret : WORD ;
END_VAR
VAR
  Error_T1 : SFB 4;
  Error_T2 : SFB 4;
  Adv_End_Aux : BOOL ;
  Ret_End_Aux : BOOL ;
  CHK_Aux1 : BOOL ;
  CHK_Aux2 : BOOL ;
  Error_T1_DN : BOOL ;
  Error_T2_DN : BOOL ;
  Adv_Memo : BOOL ;
  Visu_Adv_Arr : ARRAY  [0 .. 15 ] OF BOOL ;
  Visu_Ret_Arr : ARRAY  [0 .. 15 ] OF BOOL ;
  BLK_Move_Ret : INT ;
  Enable : BOOL ;
  Adv_End : BOOL ;
  Ret_End : BOOL ;
END_VAR
BEGIN
NETWORK
TITLE =
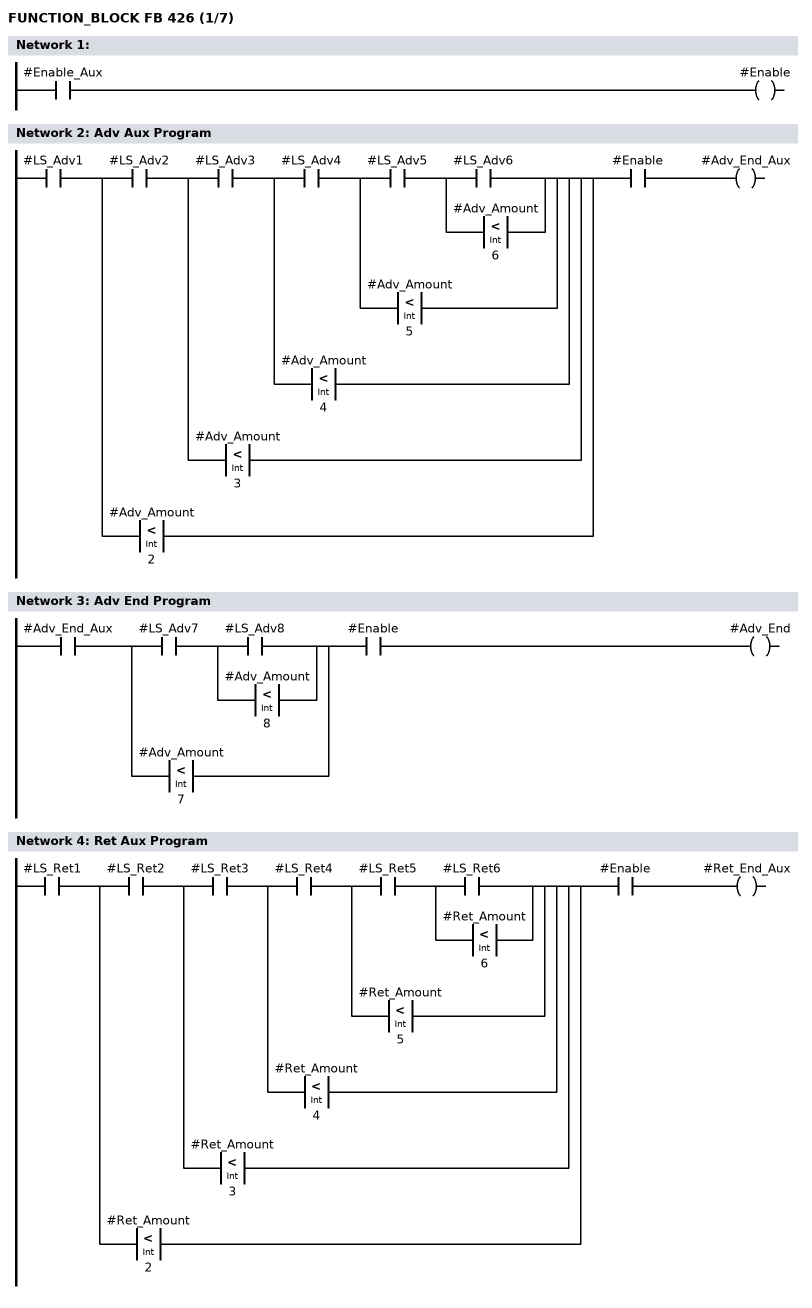

      A     #Enable_Aux;
      =     #Enable;
NETWORK
TITLE =Adv Aux Program

      A     #LS_Adv1;
      A(    ;
      A     #LS_Adv2;
      A(    ;
      A     #LS_Adv3;
      A(    ;
      A     #LS_Adv4;
      A(    ;
      A     #LS_Adv5;
      A(    ;
      O     #LS_Adv6;
      O(    ;
      L     #Adv_Amount;
      L     6;
      <I    ;
      )     ;
      )     ;
      O(    ;
      L     #Adv_Amount;
      L     5;
      <I    ;
      )     ;
      )     ;
      O(    ;
      L     #Adv_Amount;
      L     4;
      <I    ;
      )     ;
      )     ;
      O(    ;
      L     #Adv_Amount;
      L     3;
      <I    ;
      )     ;
      )     ;
      O(    ;
      L     #Adv_Amount;
      L     2;
      <I    ;
      )     ;
      )     ;
      A     #Enable;
      =     #Adv_End_Aux;
NETWORK
TITLE =Adv End Program

      A     #Adv_End_Aux;
      A(    ;
      A     #LS_Adv7;
      A(    ;
      O     #LS_Adv8;
      O(    ;
      L     #Adv_Amount;
      L     8;
      <I    ;
      )     ;
      )     ;
      O(    ;
      L     #Adv_Amount;
      L     7;
      <I    ;
      )     ;
      )     ;
      A     #Enable;
      =     #Adv_End;
NETWORK
TITLE =Ret Aux Program

      A     #LS_Ret1;
      A(    ;
      A     #LS_Ret2;
      A(    ;
      A     #LS_Ret3;
      A(    ;
      A     #LS_Ret4;
      A(    ;
      A     #LS_Ret5;
      A(    ;
      O     #LS_Ret6;
      O(    ;
      L     #Ret_Amount;
      L     6;
      <I    ;
      )     ;
      )     ;
      O(    ;
      L     #Ret_Amount;
      L     5;
      <I    ;
      )     ;
      )     ;
      O(    ;
      L     #Ret_Amount;
      L     4;
      <I    ;
      )     ;
      )     ;
      O(    ;
      L     #Ret_Amount;
      L     3;
      <I    ;
      )     ;
      )     ;
      O(    ;
      L     #Ret_Amount;
      L     2;
      <I    ;
      )     ;
      )     ;
      A     #Enable;
      =     #Ret_End_Aux;
NETWORK
TITLE =Ret End Program
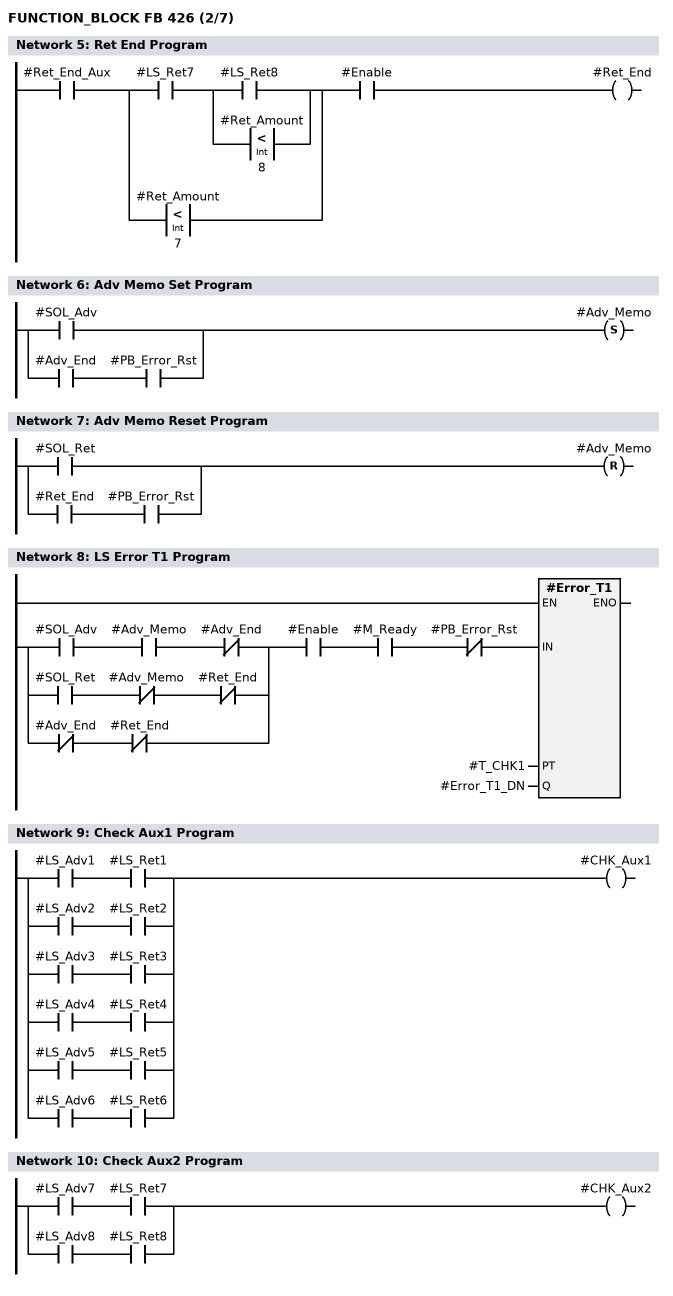

      A     #Ret_End_Aux;
      A(    ;
      A     #LS_Ret7;
      A(    ;
      O     #LS_Ret8;
      O(    ;
      L     #Ret_Amount;
      L     8;
      <I    ;
      )     ;
      )     ;
      O(    ;
      L     #Ret_Amount;
      L     7;
      <I    ;
      )     ;
      )     ;
      A     #Enable;
      =     #Ret_End;
NETWORK
TITLE =Adv Memo Set Program

      O     #SOL_Adv;
      O     ;
      A     #Adv_End;
      A     #PB_Error_Rst;
      S     #Adv_Memo;
NETWORK
TITLE =Adv Memo Reset Program

      O     #SOL_Ret;
      O     ;
      A     #Ret_End;
      A     #PB_Error_Rst;
      R     #Adv_Memo;
NETWORK
TITLE =LS Error T1 Program

      A(    ;
      A     #SOL_Adv;
      A     #Adv_Memo;
      AN    #Adv_End;
      O     ;
      A     #SOL_Ret;
      AN    #Adv_Memo;
      AN    #Ret_End;
      O     ;
      AN    #Adv_End;
      AN    #Ret_End;
      )     ;
      A     #Enable;
      A     #M_Ready;
      AN    #PB_Error_Rst;
      =     L      0.0;
      BLD   103;
      CALL #Error_T1 (
           IN                       := L      0.0,
           PT                       := #T_CHK1,
           Q                        := #Error_T1_DN);

      NOP   0;
NETWORK
TITLE =Check Aux1 Program

      A     #LS_Adv1;
      A     #LS_Ret1;
      O     ;
      A     #LS_Adv2;
      A     #LS_Ret2;
      O     ;
      A     #LS_Adv3;
      A     #LS_Ret3;
      O     ;
      A     #LS_Adv4;
      A     #LS_Ret4;
      O     ;
      A     #LS_Adv5;
      A     #LS_Ret5;
      O     ;
      A     #LS_Adv6;
      A     #LS_Ret6;
      =     #CHK_Aux1;
NETWORK
TITLE =Check Aux2 Program

      A     #LS_Adv7;
      A     #LS_Ret7;
      O     ;
      A     #LS_Adv8;
      A     #LS_Ret8;
      =     #CHK_Aux2;
NETWORK
TITLE =LS Error T2 Program
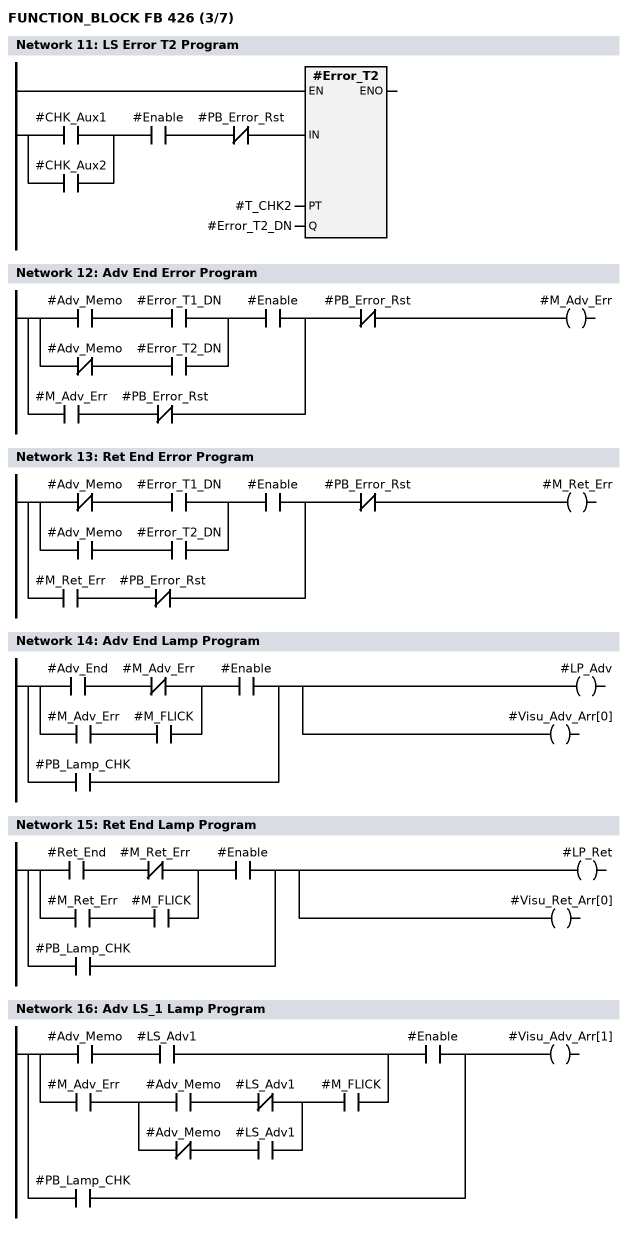

      A(    ;
      O     #CHK_Aux1;
      O     #CHK_Aux2;
      )     ;
      A     #Enable;
      AN    #PB_Error_Rst;
      =     L      0.0;
      BLD   103;
      CALL #Error_T2 (
           IN                       := L      0.0,
           PT                       := #T_CHK2,
           Q                        := #Error_T2_DN);

      NOP   0;
NETWORK
TITLE =Adv End Error Program

      A(    ;
      A(    ;
      A     #Adv_Memo;
      A     #Error_T1_DN;
      O     ;
      AN    #Adv_Memo;
      A     #Error_T2_DN;
      )     ;
      A     #Enable;
      O     ;
      A     #M_Adv_Err;
      AN    #PB_Error_Rst;
      )     ;
      AN    #PB_Error_Rst;
      =     #M_Adv_Err;
NETWORK
TITLE =Ret End Error Program

      A(    ;
      A(    ;
      AN    #Adv_Memo;
      A     #Error_T1_DN;
      O     ;
      A     #Adv_Memo;
      A     #Error_T2_DN;
      )     ;
      A     #Enable;
      O     ;
      A     #M_Ret_Err;
      AN    #PB_Error_Rst;
      )     ;
      AN    #PB_Error_Rst;
      =     #M_Ret_Err;
NETWORK
TITLE =Adv End Lamp Program

      A(    ;
      A     #Adv_End;
      AN    #M_Adv_Err;
      O     ;
      A     #M_Adv_Err;
      A     #M_FLICK;
      )     ;
      A     #Enable;
      O     #PB_Lamp_CHK;
      =     #LP_Adv;
      =     #Visu_Adv_Arr[0];
NETWORK
TITLE =Ret End Lamp Program

      A(    ;
      A     #Ret_End;
      AN    #M_Ret_Err;
      O     ;
      A     #M_Ret_Err;
      A     #M_FLICK;
      )     ;
      A     #Enable;
      O     #PB_Lamp_CHK;
      =     #LP_Ret;
      =     #Visu_Ret_Arr[0];
NETWORK
TITLE =Adv LS_1 Lamp Program

      A(    ;
      A     #Adv_Memo;
      A     #LS_Adv1;
      O     ;
      A     #M_Adv_Err;
      A(    ;
      A     #Adv_Memo;
      AN    #LS_Adv1;
      O     ;
      AN    #Adv_Memo;
      A     #LS_Adv1;
      )     ;
      A     #M_FLICK;
      )     ;
      A     #Enable;
      O     #PB_Lamp_CHK;
      =     #Visu_Adv_Arr[1];
NETWORK
TITLE =Adv LS_2 Lamp Program
//
//
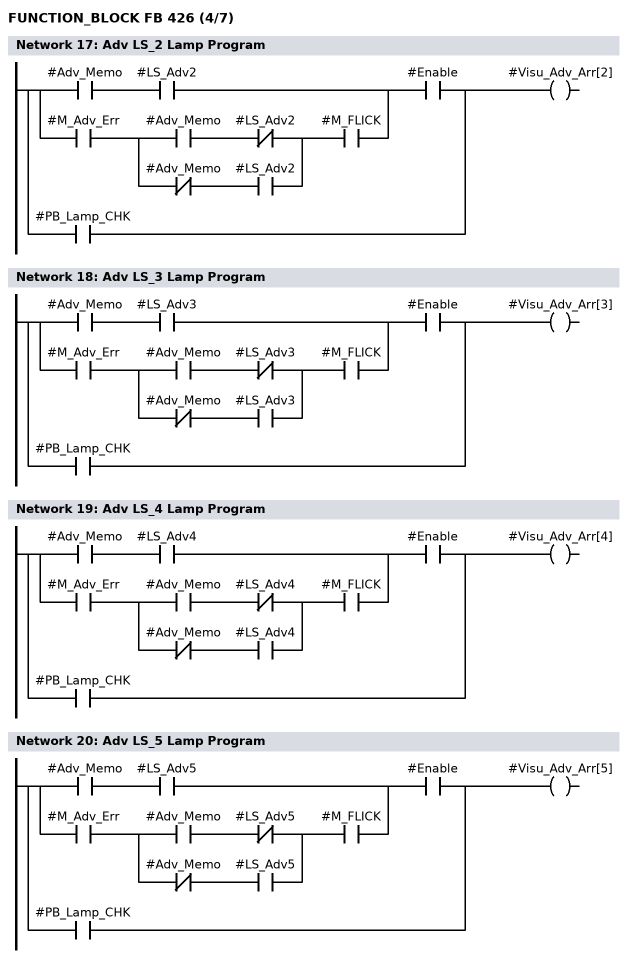
      A(    ;
      A     #Adv_Memo;
      A     #LS_Adv2;
      O     ;
      A     #M_Adv_Err;
      A(    ;
      A     #Adv_Memo;
      AN    #LS_Adv2;
      O     ;
      AN    #Adv_Memo;
      A     #LS_Adv2;
      )     ;
      A     #M_FLICK;
      )     ;
      A     #Enable;
      O     #PB_Lamp_CHK;
      =     #Visu_Adv_Arr[2];
NETWORK
TITLE =Adv LS_3 Lamp Program
//
//
      A(    ;
      A     #Adv_Memo;
      A     #LS_Adv3;
      O     ;
      A     #M_Adv_Err;
      A(    ;
      A     #Adv_Memo;
      AN    #LS_Adv3;
      O     ;
      AN    #Adv_Memo;
      A     #LS_Adv3;
      )     ;
      A     #M_FLICK;
      )     ;
      A     #Enable;
      O     #PB_Lamp_CHK;
      =     #Visu_Adv_Arr[3];
NETWORK
TITLE =Adv LS_4 Lamp Program
//
//
      A(    ;
      A     #Adv_Memo;
      A     #LS_Adv4;
      O     ;
      A     #M_Adv_Err;
      A(    ;
      A     #Adv_Memo;
      AN    #LS_Adv4;
      O     ;
      AN    #Adv_Memo;
      A     #LS_Adv4;
      )     ;
      A     #M_FLICK;
      )     ;
      A     #Enable;
      O     #PB_Lamp_CHK;
      =     #Visu_Adv_Arr[4];
NETWORK
TITLE =Adv LS_5 Lamp Program
//
//
      A(    ;
      A     #Adv_Memo;
      A     #LS_Adv5;
      O     ;
      A     #M_Adv_Err;
      A(    ;
      A     #Adv_Memo;
      AN    #LS_Adv5;
      O     ;
      AN    #Adv_Memo;
      A     #LS_Adv5;
      )     ;
      A     #M_FLICK;
      )     ;
      A     #Enable;
      O     #PB_Lamp_CHK;
      =     #Visu_Adv_Arr[5];
NETWORK
TITLE =Adv LS_6 Lamp Program
//
//
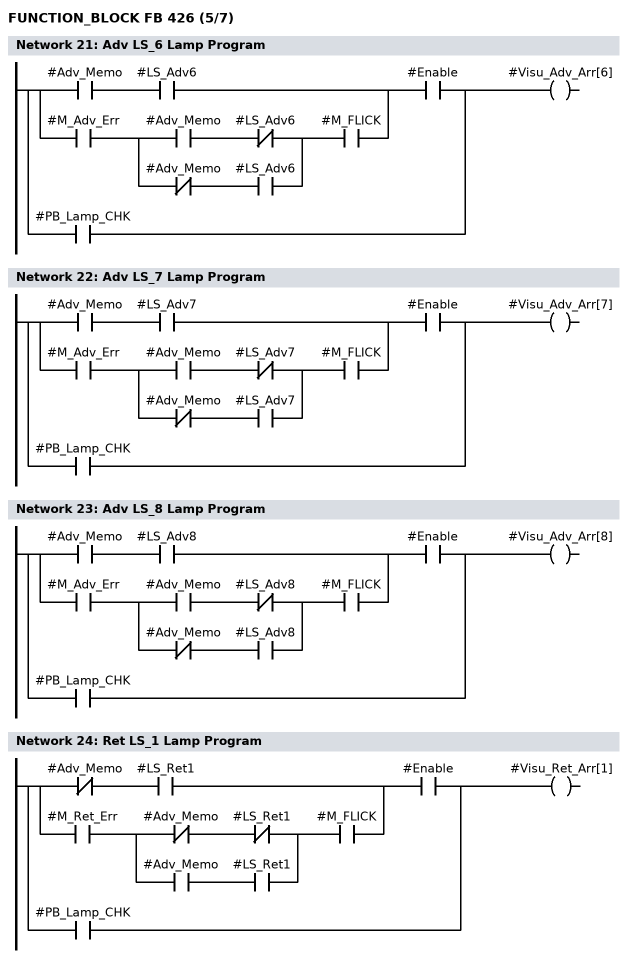
      A(    ;
      A     #Adv_Memo;
      A     #LS_Adv6;
      O     ;
      A     #M_Adv_Err;
      A(    ;
      A     #Adv_Memo;
      AN    #LS_Adv6;
      O     ;
      AN    #Adv_Memo;
      A     #LS_Adv6;
      )     ;
      A     #M_FLICK;
      )     ;
      A     #Enable;
      O     #PB_Lamp_CHK;
      =     #Visu_Adv_Arr[6];
NETWORK
TITLE =Adv LS_7 Lamp Program
//
//
      A(    ;
      A     #Adv_Memo;
      A     #LS_Adv7;
      O     ;
      A     #M_Adv_Err;
      A(    ;
      A     #Adv_Memo;
      AN    #LS_Adv7;
      O     ;
      AN    #Adv_Memo;
      A     #LS_Adv7;
      )     ;
      A     #M_FLICK;
      )     ;
      A     #Enable;
      O     #PB_Lamp_CHK;
      =     #Visu_Adv_Arr[7];
NETWORK
TITLE =Adv LS_8 Lamp Program
//
//
      A(    ;
      A     #Adv_Memo;
      A     #LS_Adv8;
      O     ;
      A     #M_Adv_Err;
      A(    ;
      A     #Adv_Memo;
      AN    #LS_Adv8;
      O     ;
      AN    #Adv_Memo;
      A     #LS_Adv8;
      )     ;
      A     #M_FLICK;
      )     ;
      A     #Enable;
      O     #PB_Lamp_CHK;
      =     #Visu_Adv_Arr[8];
NETWORK
TITLE =Ret LS_1 Lamp Program
//
//
      A(    ;
      AN    #Adv_Memo;
      A     #LS_Ret1;
      O     ;
      A     #M_Ret_Err;
      A(    ;
      AN    #Adv_Memo;
      AN    #LS_Ret1;
      O     ;
      A     #Adv_Memo;
      A     #LS_Ret1;
      )     ;
      A     #M_FLICK;
      )     ;
      A     #Enable;
      O     #PB_Lamp_CHK;
      =     #Visu_Ret_Arr[1];
NETWORK
TITLE =Ret LS_2 Lamp Program
//
//
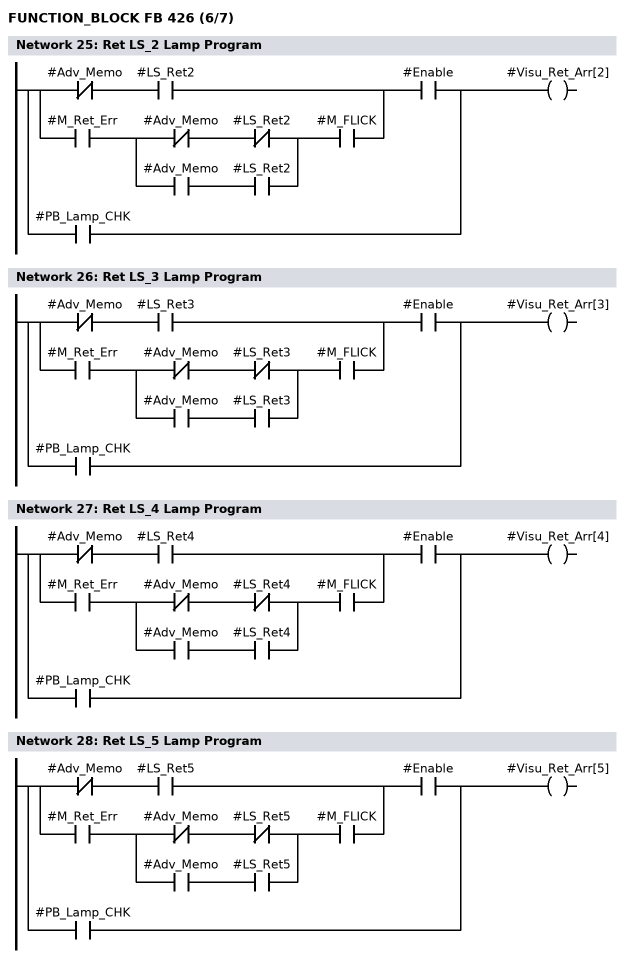
      A(    ;
      AN    #Adv_Memo;
      A     #LS_Ret2;
      O     ;
      A     #M_Ret_Err;
      A(    ;
      AN    #Adv_Memo;
      AN    #LS_Ret2;
      O     ;
      A     #Adv_Memo;
      A     #LS_Ret2;
      )     ;
      A     #M_FLICK;
      )     ;
      A     #Enable;
      O     #PB_Lamp_CHK;
      =     #Visu_Ret_Arr[2];
NETWORK
TITLE =Ret LS_3 Lamp Program
//
//
      A(    ;
      AN    #Adv_Memo;
      A     #LS_Ret3;
      O     ;
      A     #M_Ret_Err;
      A(    ;
      AN    #Adv_Memo;
      AN    #LS_Ret3;
      O     ;
      A     #Adv_Memo;
      A     #LS_Ret3;
      )     ;
      A     #M_FLICK;
      )     ;
      A     #Enable;
      O     #PB_Lamp_CHK;
      =     #Visu_Ret_Arr[3];
NETWORK
TITLE =Ret LS_4 Lamp Program
//
//
      A(    ;
      AN    #Adv_Memo;
      A     #LS_Ret4;
      O     ;
      A     #M_Ret_Err;
      A(    ;
      AN    #Adv_Memo;
      AN    #LS_Ret4;
      O     ;
      A     #Adv_Memo;
      A     #LS_Ret4;
      )     ;
      A     #M_FLICK;
      )     ;
      A     #Enable;
      O     #PB_Lamp_CHK;
      =     #Visu_Ret_Arr[4];
NETWORK
TITLE =Ret LS_5 Lamp Program
//
//
      A(    ;
      AN    #Adv_Memo;
      A     #LS_Ret5;
      O     ;
      A     #M_Ret_Err;
      A(    ;
      AN    #Adv_Memo;
      AN    #LS_Ret5;
      O     ;
      A     #Adv_Memo;
      A     #LS_Ret5;
      )     ;
      A     #M_FLICK;
      )     ;
      A     #Enable;
      O     #PB_Lamp_CHK;
      =     #Visu_Ret_Arr[5];
NETWORK
TITLE =Ret LS_6 Lamp Program
//
//
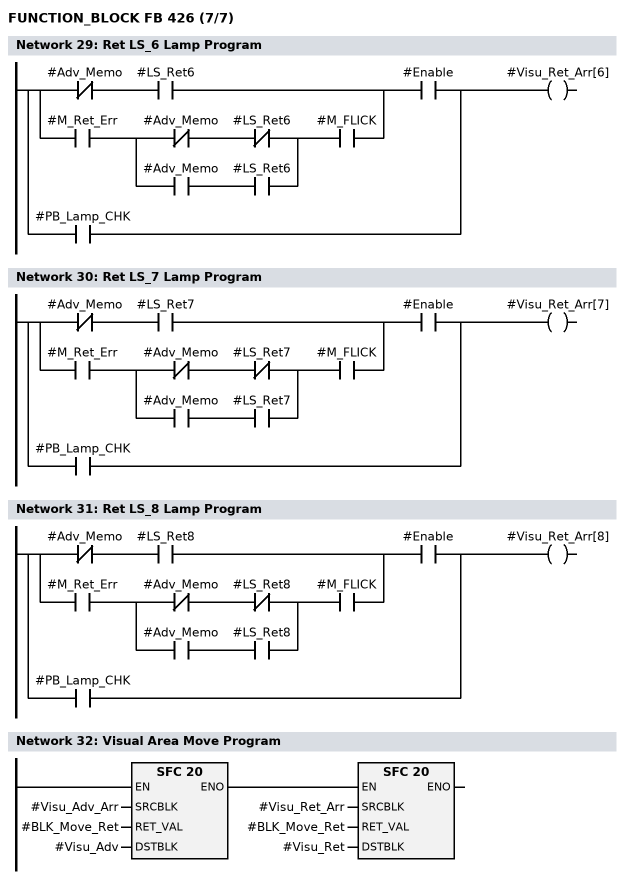
      A(    ;
      AN    #Adv_Memo;
      A     #LS_Ret6;
      O     ;
      A     #M_Ret_Err;
      A(    ;
      AN    #Adv_Memo;
      AN    #LS_Ret6;
      O     ;
      A     #Adv_Memo;
      A     #LS_Ret6;
      )     ;
      A     #M_FLICK;
      )     ;
      A     #Enable;
      O     #PB_Lamp_CHK;
      =     #Visu_Ret_Arr[6];
NETWORK
TITLE =Ret LS_7 Lamp Program
//
//
      A(    ;
      AN    #Adv_Memo;
      A     #LS_Ret7;
      O     ;
      A     #M_Ret_Err;
      A(    ;
      AN    #Adv_Memo;
      AN    #LS_Ret7;
      O     ;
      A     #Adv_Memo;
      A     #LS_Ret7;
      )     ;
      A     #M_FLICK;
      )     ;
      A     #Enable;
      O     #PB_Lamp_CHK;
      =     #Visu_Ret_Arr[7];
NETWORK
TITLE =Ret LS_8 Lamp Program
//
//
      A(    ;
      AN    #Adv_Memo;
      A     #LS_Ret8;
      O     ;
      A     #M_Ret_Err;
      A(    ;
      AN    #Adv_Memo;
      AN    #LS_Ret8;
      O     ;
      A     #Adv_Memo;
      A     #LS_Ret8;
      )     ;
      A     #M_FLICK;
      )     ;
      A     #Enable;
      O     #PB_Lamp_CHK;
      =     #Visu_Ret_Arr[8];
NETWORK
TITLE =Visual Area Move Program

      A(    ;
      CALL SFC   20 (
           SRCBLK                   := #Visu_Adv_Arr,
           RET_VAL                  := #BLK_Move_Ret,
           DSTBLK                   := #Visu_Adv);
      A     BR;
      )     ;
      JNB   _001;
      CALL SFC   20 (
           SRCBLK                   := #Visu_Ret_Arr,
           RET_VAL                  := #BLK_Move_Ret,
           DSTBLK                   := #Visu_Ret);
_001: NOP   0;
END_FUNCTION_BLOCK

FUNCTION_BLOCK FB 470
TITLE =HMI Body Type Modify Variables Program
AUTHOR : HMC
FAMILY : HMI
NAME : HMI
VERSION : 1.0


VAR_INPUT
  Station : INT ;
  HMI_Disp_DB : INT ;
  HMI_Disp_Add : INT ;
  CType_DB : INT ;
  CType_Start_Add : INT ;
  Byte_per_Stn : INT ;
  M_Modify_OK : BOOL ;
  SS_CCR_On : BOOL ;
  PB_Set : BOOL ;
  PB_Reset : BOOL ;
END_VAR
VAR_OUTPUT
  LP_CCR_On : BOOL ;
  LP_Modify_On : BOOL ;
END_VAR
VAR
  Source_Data : WORD ;
  Modify_Data : WORD ;
  Pre_Station : INT ;
  Station_PLS : BOOL ;
  Source_Add : INT ;
  SFC20_Ret : INT ;
  Fill_Source : WORD ;
END_VAR
VAR_TEMP
  Source_Area : ANY ;
  Modify_Area : ANY ;
END_VAR
BEGIN
NETWORK
TITLE =FAC On Lamp Program

      A     #SS_CCR_On;
      =     #LP_CCR_On;
NETWORK
TITLE =Operation Pulse

      L     #Station; // Station Select Data
      L     0; // Is Not Zero
      <>I   ;
      JNB   _End; // Jump to End
NETWORK
TITLE =Modify On Lamp Program
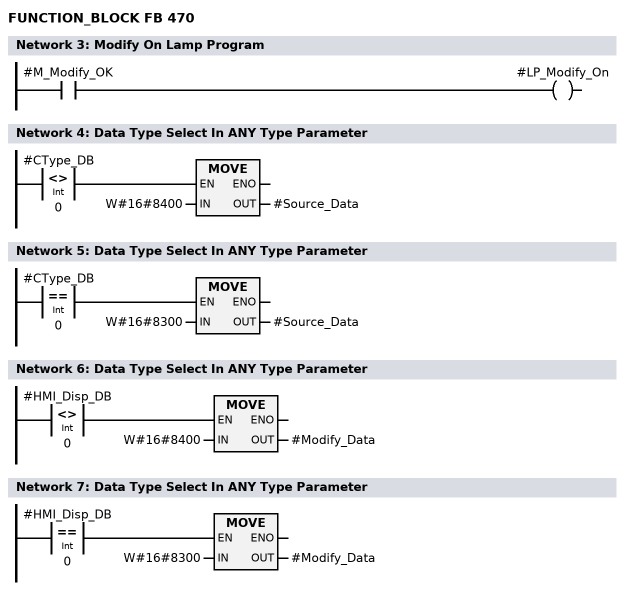

      A     #M_Modify_OK;
      =     #LP_Modify_On;
NETWORK
TITLE =Data Type Select In ANY Type Parameter

      A(    ; // If Source DB is Not Zero
      L     #CType_DB;
      L     0;
      <>I   ;
      )     ;
      JNB   _B01; // Jump to Next Step
      L     W#16#8400; // Load "8400" _ Means "DB Area"
      T     #Source_Data; // Transfer to Data_Type
_B01: NOP   0;
NETWORK
TITLE =Data Type Select In ANY Type Parameter

      A(    ; // If DB_NO is Zero
      L     #CType_DB;
      L     0;
      ==I   ;
      )     ;
      JNB   _B02; // Jump to Next Step
      L     W#16#8300; // Load "8300" _ Means "Bit Memory Area"
      T     #Source_Data; // Transfer to Data_Type
_B02: NOP   0;
NETWORK
TITLE =Data Type Select In ANY Type Parameter

      A(    ; // If Source DB is Not Zero
      L     #HMI_Disp_DB;
      L     0;
      <>I   ;
      )     ;
      JNB   _B03; // Jump to Next Step
      L     W#16#8400; // Load "8400" _ Means "DB Area"
      T     #Modify_Data; // Transfer to Data_Type
_B03: NOP   0;
NETWORK
TITLE =Data Type Select In ANY Type Parameter

      A(    ; // If DB_NO is Zero
      L     #HMI_Disp_DB;
      L     0;
      ==I   ;
      )     ;
      JNB   _B04; // Jump to Next Step
      L     W#16#8300; // Load "8300" _ Means "Bit Memory Area"
      T     #Modify_Data; // Transfer to Data_Type
_B04: NOP   0;
NETWORK
TITLE =Source Area Start Address Calculate Porgram

      L     #Station; // Station Amount - 1
      L     1;
      -I    ;
      L     #Byte_per_Stn; // Multi Length Per Station
      *I    ;
      L     #CType_Start_Add;
      +I    ;
      T     #Source_Add;
NETWORK
TITLE =Make a "ANY" Type Data

      LAR1  P##Source_Area; // Load 1st Station Address of ANY Pointer In "AR1"

      L     B#16#10; // Load Syntax ID For S7 "10"
      T     LB [AR1,P#0.0]; // Transfer ID to the ANY Pointer

      L     B#16#2; // Load Data Type _ "2" means "BYTE"
      T     LB [AR1,P#1.0]; // Transfer Data Type to the ANY Pointer

      L     #Byte_per_Stn; // Load the Length of Source Data
      T     LW [AR1,P#2.0]; // Transfer the Numbers to the ANY Pointer

      L     #CType_DB; // Load DB Number _ "0" means don't use "DB"
      T     LW [AR1,P#4.0]; // Transfer the Numbers to the ANY Pointer

      L     #Source_Data; // Load Data Type _ "83" means "Bit Memory" Area
      T     LW [AR1,P#6.0]; //                  "84" means "DB" Area

      L     #Source_Add; // Load Start Address
      SLW   3; // Shift Left Word _ "3" Bit
      T     LW [AR1,P#8.0]; // Transfer the Address to the ANY Pointer

      LAR1  P##Modify_Area; // Load 2nd Station Address of ANY Pointer In "AR1"

      L     B#16#10; //Load Syntax ID For S7 "10"
      T     LB [AR1,P#0.0]; //Load Syntax ID For S7 "10"

      L     B#16#2; //  Load Data Type _ "2" means "BYTE"
      T     LB [AR1,P#1.0]; // Transfer Data Type to the ANY Pointer

      L     #Byte_per_Stn; // Load the Length of Target Data
      T     LW [AR1,P#2.0]; // Transfer the Numbers to the ANY Pointer

      L     #HMI_Disp_DB; // Load DB Number _ "0" means don't use "DB"
      T     LW [AR1,P#4.0]; // Transfer the Numbers to the ANY Pointer

      L     #Modify_Data; // Load Data Type _ "83" means "Bit Memory" Area
      T     LW [AR1,P#6.0]; //                  "84" means "DB" Area

      L     #HMI_Disp_Add; //  Load Start Address
      SLW   3; // Shift Left Word _ "3" Bit
      T     LW [AR1,P#8.0]; // Transfer the Address to the ANY Pointer

NETWORK
TITLE =Copy To Modify Area Program

      L     #Station;
      L     #Pre_Station;
      <>I   ;
      JNB   _B05;
NETWORK
TITLE =Copy To Previous Station No Program

      L     #Station;
      T     #Pre_Station;
NETWORK
TITLE =Block Move to Modify Area


      CALL SFC   20 (
           SRCBLK                   := #Source_Area,
           RET_VAL                  := #SFC20_Ret,
           DSTBLK                   := #Modify_Area);
_B05: NOP   0;
NETWORK
TITLE =Data Clear Program

      A     #M_Modify_OK;
      A     #PB_Reset;
      JNB   _B06;
NETWORK
TITLE =Clear Source Data Area


      CALL SFC   21 (
           BVAL                     := #Fill_Source,// "Zero"
           RET_VAL                  := #SFC20_Ret,
           BLK                      := #Source_Area);// Transfer to First Station Area

NETWORK
TITLE =Clear Source Data Area


      CALL SFC   21 (
           BVAL                     := #Fill_Source,// "Zero"
           RET_VAL                  := #SFC20_Ret,
           BLK                      := #Modify_Area);// Transfer to First Station Area
_B06: NOP   0;
NETWORK
TITLE =Data Clear Program

      A     #M_Modify_OK;
      A     #PB_Set;
      JNB   _B07;
NETWORK
TITLE =Block Move to Modify Area


      CALL SFC   20 (
           SRCBLK                   := #Modify_Area,
           RET_VAL                  := #SFC20_Ret,
           DSTBLK                   := #Source_Area);
_B07: NOP   0;
NETWORK
TITLE =


_End: NOP   0;

END_FUNCTION_BLOCK

FUNCTION_BLOCK FB 500
TITLE =CYCLE TIME CHECK
VERSION : 0.1


VAR_INPUT
  CYCLE_UP : BOOL ;
  CYCLE_RST : BOOL ;
END_VAR
VAR_OUTPUT
  CURRENT_CT : INT ;
  PREVIOUS_CT : INT ;
END_VAR
VAR
  CURRENT : INT ;
  PREVIOUS : INT ;
  CYCLE_UP_PLS : BOOL ;
  CYCLE_RST_PLS : BOOL ;
  CYCLE_OVER_PLS : BOOL ;
END_VAR
BEGIN
NETWORK
TITLE =CURRENT TIME CHK
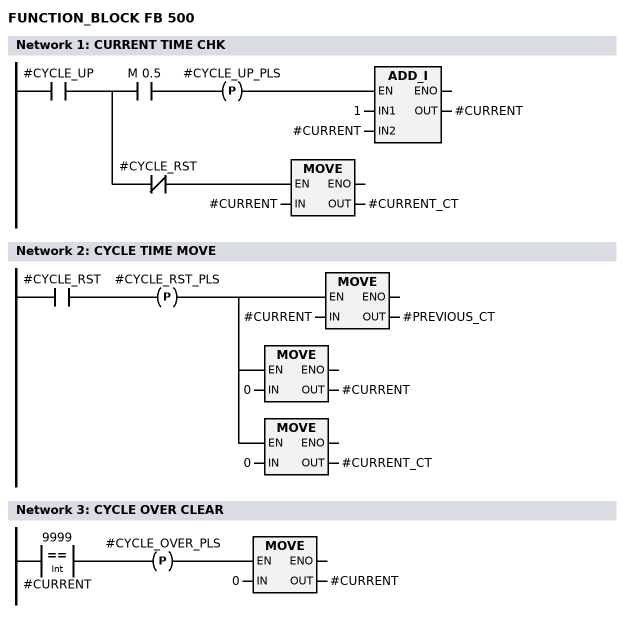

      A     #CYCLE_UP;
      =     L      0.0;
      A     L      0.0;
      A     M      0.5;
      FP    #CYCLE_UP_PLS;
      JNB   _001;
      L     1;
      L     #CURRENT;
      +I    ;
      T     #CURRENT;
_001: NOP   0;
      A     L      0.0;
      AN    #CYCLE_RST;
      JNB   _002;
      L     #CURRENT;
      T     #CURRENT_CT;
_002: NOP   0;
NETWORK
TITLE =CYCLE TIME MOVE

      A     #CYCLE_RST;
      FP    #CYCLE_RST_PLS;
      =     L      0.0;
      A     L      0.0;
      JNB   _003;
      L     #CURRENT;
      T     #PREVIOUS_CT;
_003: NOP   0;
      A     L      0.0;
      JNB   _004;
      L     0;
      T     #CURRENT;
_004: NOP   0;
      A     L      0.0;
      JNB   _005;
      L     0;
      T     #CURRENT_CT;
_005: NOP   0;
NETWORK
TITLE =CYCLE OVER CLEAR

      A(    ;
      L     9999;
      L     #CURRENT;
      ==I   ;
      )     ;
      FP    #CYCLE_OVER_PLS;
      JNB   _006;
      L     0;
      T     #CURRENT;
_006: NOP   0;
END_FUNCTION_BLOCK

FUNCTION FC 502 : VOID
TITLE =
VERSION : 1.0


VAR_INPUT
  IN0 : INT ;
  IN1 : WORD ;
  IN2 : INT ;
  IN3 : WORD ;
END_VAR
VAR_TEMP
  TEMP4 : INT ;
  TEMP5 : DATE_AND_TIME ;
  TEMP6 : INT ;
END_VAR
BEGIN
NETWORK
TITLE =

      L     #IN0;
      T     #TEMP4;
      OPN   DB [#TEMP4];
      L     0;
      T     DBW   92;
      NOP   0;
NETWORK
TITLE =

      A(    ;
      L     1090;
      T     DBW   94;
      SET   ;
      SAVE  ;
      CLR   ;
      A     BR;
      )     ;
      JNB   _001;
      L     DBW   94;
      L     10;
      -I    ;
      T     DBW   96;
_001: NOP   0;
NETWORK
TITLE =

M003: L     100;
      L     DBW   92;
      ==I   ;
      JC    M002;
      L     DBW   94;
      SLW   3;
      LAR1  ;
      L     DBW   96;
      SLW   3;
      LAR2  ;
      L     DBD [AR2,P#0.0];
      T     DBD [AR1,P#0.0];
      L     DBD [AR2,P#4.0];
      T     DBD [AR1,P#4.0];
      L     DBW [AR2,P#8.0];
      T     DBW [AR1,P#8.0];
      L     DBW   94;
      L     10;
      -I    ;
      T     DBW   94;
      L     DBW   96;
      L     10;
      -I    ;
      T     DBW   96;
      L     1;
      L     DBW   92;
      +I    ;
      T     DBW   92;
      JP    M003;
M002: NOP   0;
      LAR1  P#0.0;
NETWORK
TITLE =

      CALL SFC    1 (
           RET_VAL                  := #TEMP6,
           OUT0                     := #TEMP5);
      NOP   0;
NETWORK
TITLE =

      LAR2  P#0.0;
      L     #IN1;
      T     DBW [AR1,P#100.0];
      LAR1  P##TEMP5;
      L     LB [AR1,P#2.0];
      T     DBB [AR2,P#102.0];
      L     LB [AR1,P#3.0];
      T     DBB [AR2,P#103.0];
      L     LB [AR1,P#4.0];
      T     DBB [AR2,P#104.0];
      L     LB [AR1,P#5.0];
      T     DBB [AR2,P#105.0];
      L     #IN2;
      T     DBW [AR2,P#106.0];
      L     #IN3;
      T     DBW [AR2,P#108.0];
      NOP   0;
END_FUNCTION

FUNCTION FC 503 : VOID
TITLE =
VERSION : 0.1


VAR_INPUT
  IN0 : INT ;
  IN1 : INT ;
  IN2 : INT ;
  IN3 : BYTE ;
END_VAR
VAR_TEMP
  TEMP4 : ANY ;
  TEMP5 : INT ;
  TEMP6 : INT ;
  TEMP7 : INT ;
  TEMP8 : BYTE ;
  TEMP9 : INT ;
END_VAR
BEGIN
NETWORK
TITLE =

      L     #IN0;
      T     #TEMP5;
      L     #IN1;
      T     #TEMP6;
      L     #IN2;
      T     #TEMP7;
      L     #IN3;
      T     #TEMP8;
      OPN   DB [#TEMP5];
      LAR1  P##TEMP4;
      L     B#16#10;
      T     LB [AR1,P#0.0];
      L     B#16#2;
      T     LB [AR1,P#1.0];
      L     #TEMP6;
      T     LW [AR1,P#2.0];
      L     #TEMP5;
      T     LW [AR1,P#4.0];
      L     W#16#8400;
      T     LW [AR1,P#6.0];
      L     #TEMP7;
      SLW   3;
      T     LW [AR1,P#8.0];
      CALL SFC   21 (
           BVAL                     := #TEMP8,
           RET_VAL                  := #TEMP9,
           BLK                      := #TEMP4);
      NOP   0;
END_FUNCTION

FUNCTION FC 504 : VOID
TITLE =
VERSION : 0.1


VAR_INPUT
  IN0 : INT ;
  IN1 : INT ;
  IN2 : INT ;
  IN3 : INT ;
  IN4 : INT ;
END_VAR
VAR_TEMP
  TEMP5 : ANY ;
  TEMP6 : ANY ;
  TEMP7 : INT ;
  TEMP8 : INT ;
  TEMP9 : INT ;
  TEMP10 : INT ;
  TEMP11 : INT ;
  TEMP12 : INT ;
END_VAR
BEGIN
NETWORK
TITLE =

      L     #IN0;
      T     #TEMP7;
      L     #IN2;
      T     #TEMP8;
      L     #IN1;
      T     #TEMP9;
      L     #IN3;
      T     #TEMP10;
      L     #IN4;
      T     #TEMP11;
      OPN   DB [#TEMP7];
      LAR1  P##TEMP5;
      L     B#16#10;
      T     LB [AR1,P#0.0];
      L     B#16#2;
      T     LB [AR1,P#1.0];
      L     #TEMP8;
      T     LW [AR1,P#2.0];
      L     #TEMP7;
      T     LW [AR1,P#4.0];
      L     W#16#8400;
      T     LW [AR1,P#6.0];
      L     #TEMP9;
      SLW   3;
      T     LW [AR1,P#8.0];
      LAR2  P##TEMP6;
      L     B#16#10;
      T     LB [AR2,P#0.0];
      L     B#16#2;
      T     LB [AR2,P#1.0];
      L     #IN2;
      T     LW [AR2,P#2.0];
      L     #TEMP10;
      T     LW [AR2,P#4.0];
      L     W#16#8400;
      T     LW [AR2,P#6.0];
      L     #TEMP11;
      SLW   3;
      T     LW [AR2,P#8.0];
      CALL SFC   20 (
           SRCBLK                   := #TEMP5,
           RET_VAL                  := #TEMP12,
           DSTBLK                   := #TEMP6);
      NOP   0;
END_FUNCTION

FUNCTION FC 505 : VOID
TITLE =
VERSION : 0.1


VAR_INPUT
  IN0 : INT ;
  IN1 : INT ;
END_VAR
VAR_TEMP
  TEMP2 : INT ;
  TEMP3 : INT ;
  TEMP4 : DATE_AND_TIME ;
  TEMP5 : DATE_AND_TIME ;
  TEMP6 : INT ;
  TEMP7 : INT ;
  TEMP8 : BOOL ;
END_VAR
BEGIN
NETWORK
TITLE =

      L     #IN1;
      T     #TEMP3;
      L     #IN0;
      T     #TEMP2;
      OPN   DB [#TEMP2];
      OPN   DI [#TEMP3];
      LAR1  P#0.0;
      LAR2  P#0.0;
NETWORK
TITLE =

      CALL SFC    1 (
           RET_VAL                  := #TEMP6,
           OUT0                     := #TEMP4);
      NOP   0;
NETWORK
TITLE =

      LAR1  P#0.0;
      LAR2  P#0.0;
      LAR1  P##TEMP4;
      L     LB [AR1,P#0.0];
      T     DIB [AR2,P#40.0];
      L     LB [AR1,P#1.0];
      T     DIB [AR2,P#41.0];
      NOP   0;
NETWORK
TITLE =

      LAR1  P#0.0;
      LAR2  P#0.0;
      LAR2  P##TEMP5;
      L     DIB [AR1,P#40.0];
      T     LB [AR2,P#0.0];
      L     DIB [AR1,P#41.0];
      T     LB [AR2,P#1.0];
      L     DBB  962;
      T     LB [AR2,P#2.0];
      L     DBB  963;
      T     LB [AR2,P#3.0];
      L     DBB  960;
      T     LB [AR2,P#4.0];
      L     DBB  961;
      T     LB [AR2,P#5.0];
      NOP   0;
NETWORK
TITLE =
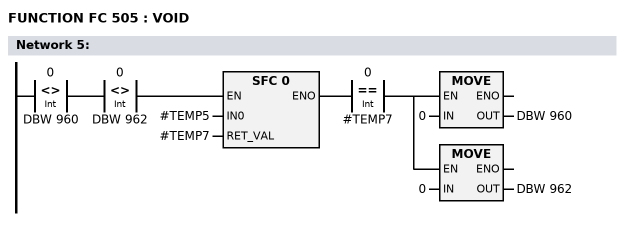

      A(    ;
      A(    ;
      L     0;
      L     DBW  960;
      <>I   ;
      )     ;
      A(    ;
      L     0;
      L     DBW  962;
      <>I   ;
      )     ;
      JNB   _001;
      CALL SFC    0 (
           IN0                      := #TEMP5,
           RET_VAL                  := #TEMP7);
_001: A     BR;
      )     ;
      A(    ;
      L     0;
      L     #TEMP7;
      ==I   ;
      )     ;
      =     L     25.0;
      A     L     25.0;
      JNB   _002;
      L     0;
      T     DBW  960;
_002: NOP   0;
      A     L     25.0;
      JNB   _003;
      L     0;
      T     DBW  962;
_003: NOP   0;
END_FUNCTION

FUNCTION_BLOCK FB 512
TITLE =Car Type Variables Program
AUTHOR : HMC
FAMILY : Car_Type
NAME : Car_Type
VERSION : 1.0


VAR_INPUT
  Stn_Vin_No : DINT ;	//Startadress Inputs from HW-Konfig
  Stn_Bt_1Word : WORD ;
  Stn_Bt_2Word : WORD ;
  Stn_Bt_3Word : WORD ;
  Stn_Bt_4Word : WORD ;
  Stn_Bt_5Word_Sp : WORD ;
  Stn_Bt_6Word_Sp : WORD ;
END_VAR
VAR_OUTPUT
  M_BType_On : BOOL ;
  M_BType_None : BOOL ;
  M_Bypass_BType : BOOL ;
  M_BType_TL : BOOL ;
  M_BType_LM : BOOL ;
  M_BType_SP1 : BOOL ;
  M_BType_SP2 : BOOL ;
  M_BType_SP3 : BOOL ;
  M_BType_DOM : BOOL ;
  M_BType_EXP : BOOL ;
  Robot_Prog_No : INT ;
END_VAR
VAR
  STN_Btype_1Arr : ARRAY  [0 .. 15 ] OF BOOL ;
  STN_Btype_2Arr : ARRAY  [0 .. 15 ] OF BOOL ;
  STN_Btype_3Arr : ARRAY  [0 .. 15 ] OF BOOL ;
  STN_Btype_4Arr : ARRAY  [0 .. 15 ] OF BOOL ;
  STN_Btype_5Arr : ARRAY  [0 .. 15 ] OF BOOL ;
  STN_Btype_6Arr : ARRAY  [0 .. 15 ] OF BOOL ;
  STN_1st_BT_On : BOOL ;
  STN_2nd_BT_On : BOOL ;
  STN_3rd_BT_On : BOOL ;
  STN_4th_BT_On : BOOL ;
  STN_5th_BT_On : BOOL ;
  STN_6th_BT_On : BOOL ;
  STN_7th_BT_On : BOOL ;
  STN_8th_BT_On : BOOL ;
  STN_9th_BT_On : BOOL ;
  STN_10th_BT_On : BOOL ;
  STN_11th_BT_On : BOOL ;
  STN_12th_BT_On : BOOL ;
  STN_1st_BT_Off : BOOL ;
  BLKMove_Ret : INT ;
  VIN_1BCD : WORD ;
  VIN_2BCD : WORD ;
  VIN_1Int : INT ;
  VIN_2Int : INT ;
END_VAR
BEGIN
NETWORK
TITLE =Station Body Type Data Change to 16-bit array

      CALL SFC   20 (
           SRCBLK                   := #Stn_Bt_1Word,
           RET_VAL                  := #BLKMove_Ret,
           DSTBLK                   := #STN_Btype_1Arr);
      NOP   0;
NETWORK
TITLE =Station Body Type Data Change to 16-bit array

      CALL SFC   20 (
           SRCBLK                   := #Stn_Bt_2Word,
           RET_VAL                  := #BLKMove_Ret,
           DSTBLK                   := #STN_Btype_2Arr);
      NOP   0;
NETWORK
TITLE =Station Body Type Data Change to 16-bit array

      CALL SFC   20 (
           SRCBLK                   := #Stn_Bt_3Word,
           RET_VAL                  := #BLKMove_Ret,
           DSTBLK                   := #STN_Btype_3Arr);
      NOP   0;
NETWORK
TITLE =Station Body Type Data Change to 16-bit array

      CALL SFC   20 (
           SRCBLK                   := #Stn_Bt_4Word,
           RET_VAL                  := #BLKMove_Ret,
           DSTBLK                   := #STN_Btype_4Arr);
      NOP   0;
NETWORK
TITLE =Station Body Type Data Change to 16-bit array

      CALL SFC   20 (
           SRCBLK                   := #Stn_Bt_5Word_Sp,
           RET_VAL                  := #BLKMove_Ret,
           DSTBLK                   := #STN_Btype_5Arr);
      NOP   0;
NETWORK
TITLE =Station Body Type Data Change to 16-bit array

      CALL SFC   20 (
           SRCBLK                   := #Stn_Bt_6Word_Sp,
           RET_VAL                  := #BLKMove_Ret,
           DSTBLK                   := #STN_Btype_6Arr);
      NOP   0;
NETWORK
TITLE =공정 1차종

      AN    OV;
      A(    ;
      O     #STN_Btype_1Arr[0];
      O     #STN_Btype_1Arr[1];
      O     #STN_Btype_1Arr[2];
      O     #STN_Btype_1Arr[3];
      O     #STN_Btype_1Arr[4];
      )     ;
      =     #STN_1st_BT_On;
NETWORK
TITLE =공정 2차종

      AN    OV;
      A(    ;
      O     #STN_Btype_1Arr[5];
      O     #STN_Btype_1Arr[6];
      O     #STN_Btype_1Arr[7];
      O     #STN_Btype_1Arr[8];
      )     ;
      =     #STN_2nd_BT_On;
NETWORK
TITLE =공정 3차종

      AN    OV;
      A(    ;
      O     #STN_Btype_1Arr[9];
      O     #STN_Btype_1Arr[10];
      )     ;
      =     #STN_3rd_BT_On;
NETWORK
TITLE =공정 4차종

      AN    OV;
      A(    ;
      O     #STN_Btype_1Arr[11];
      O     #STN_Btype_1Arr[12];
      O     #STN_Btype_1Arr[13];
      O     #STN_Btype_1Arr[14];
      O     #STN_Btype_1Arr[15];
      O     #STN_Btype_2Arr[0];
      O     #STN_Btype_2Arr[1];
      O     #STN_Btype_2Arr[2];
      O     #STN_Btype_2Arr[3];
      O     #STN_Btype_2Arr[4];
      O     #STN_Btype_2Arr[5];
      )     ;
      =     #STN_4th_BT_On;
NETWORK
TITLE =공정 5차종

      AN    OV;
      A(    ;
      O     #STN_Btype_2Arr[6];
      O     #STN_Btype_2Arr[7];
      )     ;
      =     #STN_5th_BT_On;
NETWORK
TITLE =공정 6차종

      AN    OV;
      A(    ;
      O     #STN_Btype_2Arr[8];
      O     #STN_Btype_2Arr[9];
      O     #STN_Btype_2Arr[10];
      O     #STN_Btype_2Arr[11];
      O     #STN_Btype_2Arr[12];
      O     #STN_Btype_2Arr[13];
      O     #STN_Btype_2Arr[14];
      O     #STN_Btype_2Arr[15];
      )     ;
      =     #STN_6th_BT_On;
NETWORK
TITLE =공정 7차종

      AN    OV;
      A(    ;
      O     #STN_Btype_3Arr[0];
      O     #STN_Btype_3Arr[1];
      )     ;
      =     #STN_7th_BT_On;
NETWORK
TITLE =공정 8차종

      AN    OV;
      A(    ;
      O     #STN_Btype_3Arr[2];
      O     #STN_Btype_3Arr[3];
      O     #STN_Btype_3Arr[6];
      )     ;
      =     #STN_8th_BT_On;
NETWORK
TITLE =공정 9차종

      AN    OV;
      A(    ;
      O     #STN_Btype_3Arr[4];
      O     #STN_Btype_3Arr[5];
      )     ;
      =     #STN_9th_BT_On;
NETWORK
TITLE =공정 10차종

      AN    OV;
      A(    ;
      O     #STN_Btype_3Arr[6];
      O     #STN_Btype_3Arr[7];
      )     ;
      =     #STN_10th_BT_On;
NETWORK
TITLE =공정 11차종

      AN    OV;
      A(    ;
      O     #STN_Btype_3Arr[8];
      O     #STN_Btype_3Arr[9];
      O     #STN_Btype_3Arr[10];
      O     #STN_Btype_3Arr[11];
      O     #STN_Btype_3Arr[12];
      O     #STN_Btype_3Arr[13];
      O     #STN_Btype_3Arr[14];
      O     #STN_Btype_3Arr[15];
      O     #STN_Btype_4Arr[0];
      O     #STN_Btype_4Arr[1];
      O     #STN_Btype_4Arr[2];
      O     #STN_Btype_4Arr[3];
      O     #STN_Btype_4Arr[4];
      O     #STN_Btype_4Arr[5];
      O     #STN_Btype_4Arr[6];
      O     #STN_Btype_4Arr[7];
      O     #STN_Btype_4Arr[8];
      O     #STN_Btype_4Arr[9];
      )     ;
      =     #STN_11th_BT_On;
NETWORK
TITLE =공정 차종 있음
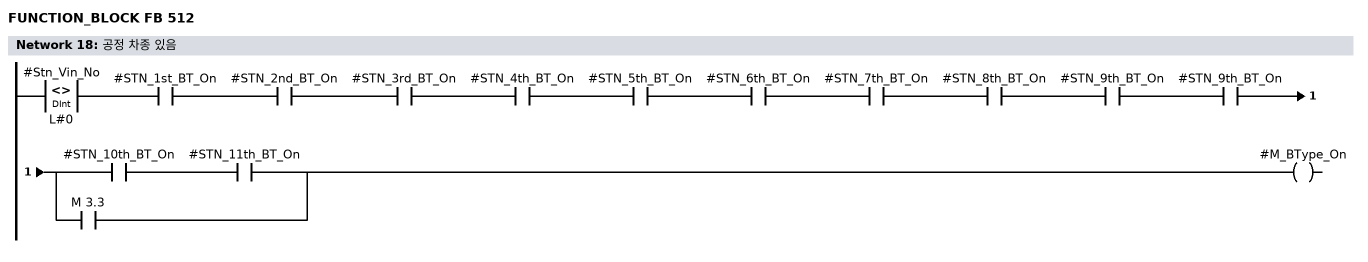

      A(    ;
      L     #Stn_Vin_No;
      L     L#0;
      <>D   ;
      )     ;
      A     #STN_1st_BT_On;
      A     #STN_2nd_BT_On;
      A     #STN_3rd_BT_On;
      A     #STN_4th_BT_On;
      A     #STN_5th_BT_On;
      A     #STN_6th_BT_On;
      A     #STN_7th_BT_On;
      A     #STN_8th_BT_On;
      A     #STN_9th_BT_On;
      A     #STN_9th_BT_On;
      A(    ;
      A     #STN_10th_BT_On;
      A     #STN_11th_BT_On;
      O     M      3.3;
      )     ;
      =     #M_BType_On;
NETWORK
TITLE =1차종 없음

      AN    OV;
      AN    #STN_Btype_1Arr[0];
      AN    #STN_Btype_1Arr[1];
      AN    #STN_Btype_1Arr[2];
      AN    #STN_Btype_1Arr[3];
      AN    #STN_Btype_1Arr[4];
      =     #STN_1st_BT_Off;
NETWORK
TITLE =공정 차종 없음
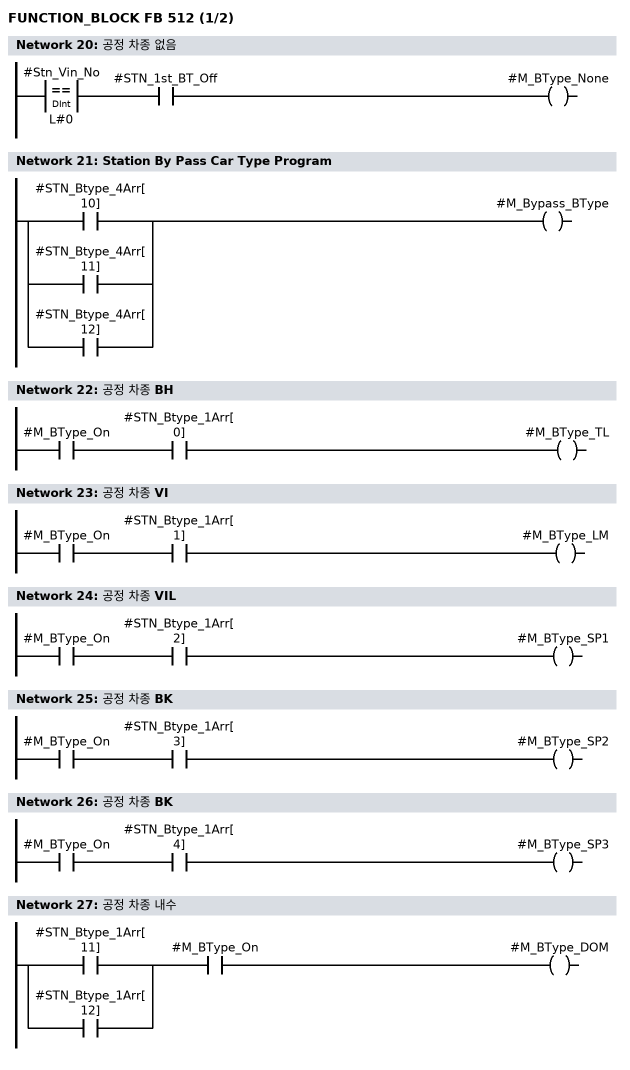

      A(    ;
      L     #Stn_Vin_No;
      L     L#0;
      ==D   ;
      )     ;
      A     #STN_1st_BT_Off;
      =     #M_BType_None;
NETWORK
TITLE =Station By Pass Car Type Program

      O     #STN_Btype_4Arr[10];
      O     #STN_Btype_4Arr[11];
      O     #STN_Btype_4Arr[12];
      =     #M_Bypass_BType;
NETWORK
TITLE =공정 차종 BH

      A     #M_BType_On;
      A     #STN_Btype_1Arr[0];
      =     #M_BType_TL;
NETWORK
TITLE =공정 차종 VI

      A     #M_BType_On;
      A     #STN_Btype_1Arr[1];
      =     #M_BType_LM;
NETWORK
TITLE =공정 차종 VIL

      A     #M_BType_On;
      A     #STN_Btype_1Arr[2];
      =     #M_BType_SP1;
NETWORK
TITLE =공정 차종 BK

      A     #M_BType_On;
      A     #STN_Btype_1Arr[3];
      =     #M_BType_SP2;
NETWORK
TITLE =공정 차종 BK

      A     #M_BType_On;
      A     #STN_Btype_1Arr[4];
      =     #M_BType_SP3;
NETWORK
TITLE =공정 차종 내수

      A(    ;
      O     #STN_Btype_1Arr[11];
      O     #STN_Btype_1Arr[12];
      )     ;
      A     #M_BType_On;
      =     #M_BType_DOM;
NETWORK
TITLE =공정 차종 수출
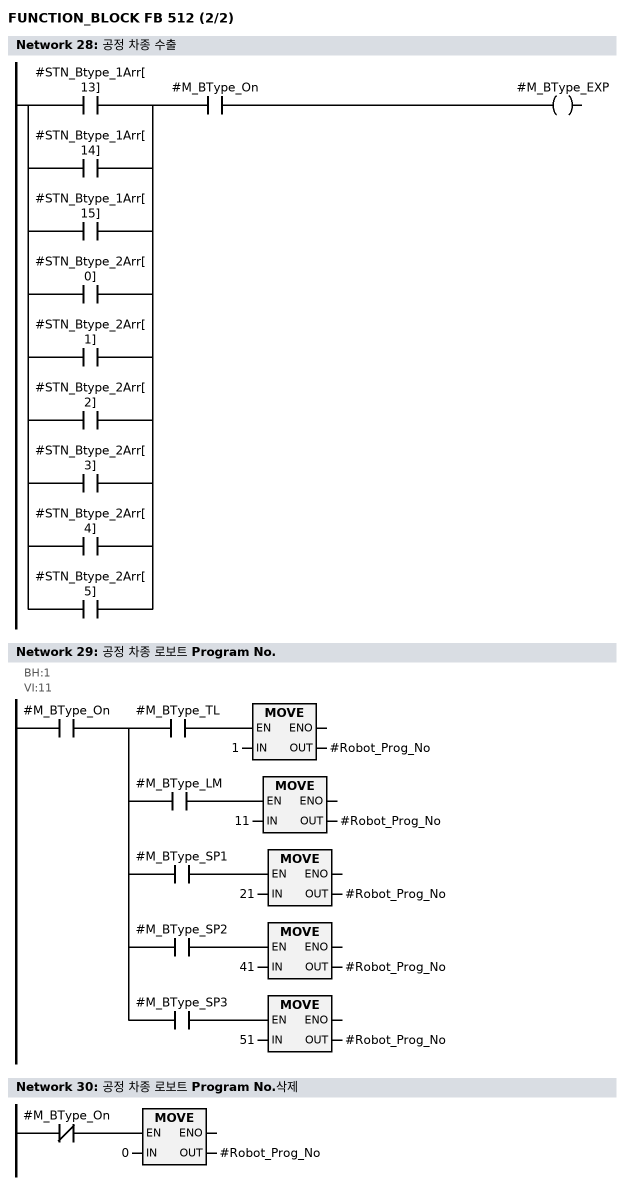

      A(    ;
      O     #STN_Btype_1Arr[13];
      O     #STN_Btype_1Arr[14];
      O     #STN_Btype_1Arr[15];
      O     #STN_Btype_2Arr[0];
      O     #STN_Btype_2Arr[1];
      O     #STN_Btype_2Arr[2];
      O     #STN_Btype_2Arr[3];
      O     #STN_Btype_2Arr[4];
      O     #STN_Btype_2Arr[5];
      )     ;
      A     #M_BType_On;
      =     #M_BType_EXP;
NETWORK
TITLE =공정 차종 로보트 Program No.
//BH:1
//VI:11
      A     #M_BType_On;
      =     L      0.0;
      A     L      0.0;
      A     #M_BType_TL;
      JNB   _001;
      L     1;
      T     #Robot_Prog_No;
_001: NOP   0;
      A     L      0.0;
      A     #M_BType_LM;
      JNB   _002;
      L     11;
      T     #Robot_Prog_No;
_002: NOP   0;
      A     L      0.0;
      A     #M_BType_SP1;
      JNB   _003;
      L     21;
      T     #Robot_Prog_No;
_003: NOP   0;
      A     L      0.0;
      A     #M_BType_SP2;
      JNB   _004;
      L     41;
      T     #Robot_Prog_No;
_004: NOP   0;
      A     L      0.0;
      A     #M_BType_SP3;
      JNB   _005;
      L     51;
      T     #Robot_Prog_No;
_005: NOP   0;
NETWORK
TITLE =공정 차종 로보트 Program No.삭제

      AN    #M_BType_On;
      JNB   _006;
      L     0;
      T     #Robot_Prog_No;
_006: NOP   0;
END_FUNCTION_BLOCK

FUNCTION_BLOCK FB 60
TITLE =
VERSION : 0.0


VAR_INPUT
  IN0 : ANY ;
  IN1 : INT ;
  IN2 : BLOCK_DB ;
END_VAR
VAR_OUTPUT
  OUT3 : WORD ;
END_VAR
VAR_IN_OUT
  IO4 : BOOL ;
  IO5 : BOOL ;
END_VAR
VAR
  STAT6 : INT ;
  STAT7 : DWORD ;
  STAT8 : DWORD ;
  STAT9 : BOOL ;
  STAT10 : BOOL ;
  STAT11 : BOOL ;
END_VAR
VAR_TEMP
  TEMP12 : BOOL ;
  TEMP13 : BOOL ;
  TEMP14 : BOOL ;
END_VAR
BEGIN
NETWORK
TITLE =

      AN    #IO4;
      JC    M002;
NETWORK
TITLE =

      L     1;
      T     #STAT6;
      NOP   0;
NETWORK
TITLE =

      LAR1  P##IN0;
      L     D [AR1,P#6.0];
      T     #STAT7;
NETWORK
TITLE =

      L     DW#16#84000000;
      T     #STAT8;
NETWORK
TITLE =

      A     #IO4;
      R     #IO4;
      R     #IO5;
NETWORK
TITLE =

M002: OPN   #IN2;

NETWORK
TITLE =

M001: L     #STAT7;
      LAR1  ;
      A      [AR1,P#0.0];
      =     #TEMP13;
NETWORK
TITLE =

      L     #STAT8;
      LAR1  ;
      A      [AR1,P#0.0];
      =     #TEMP14;
NETWORK
TITLE =
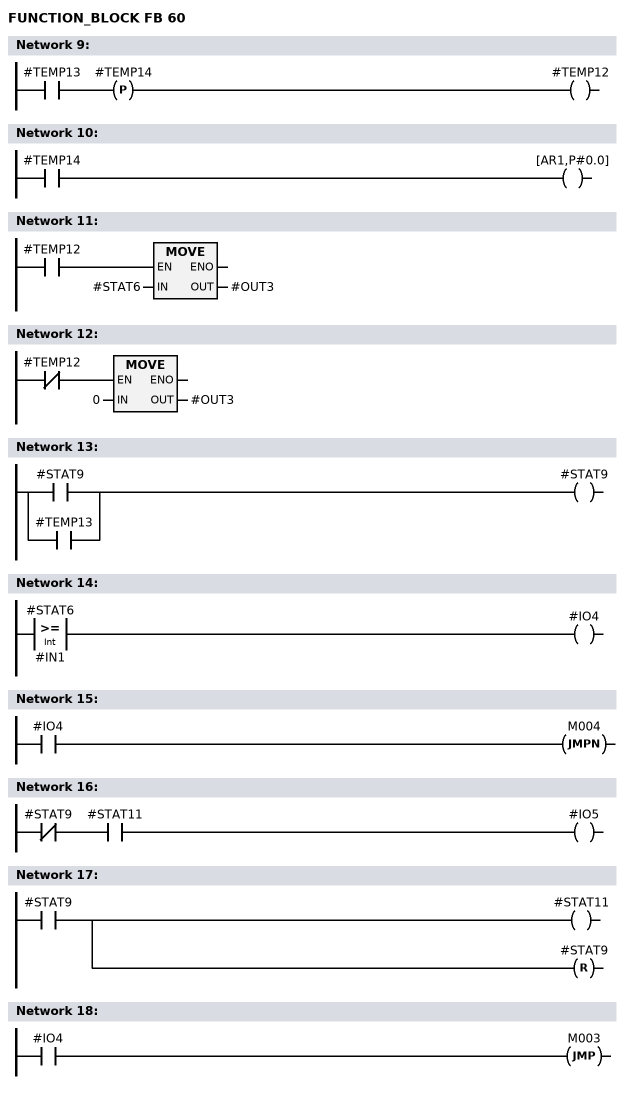

      A     #TEMP13;
      FP    #TEMP14;
      =     #TEMP12;
NETWORK
TITLE =

      A     #TEMP14;
      =      [AR1,P#0.0];
NETWORK
TITLE =

      A     #TEMP12;
      JNB   _001;
      L     #STAT6;
      T     #OUT3;
_001: NOP   0;
NETWORK
TITLE =

      AN    #TEMP12;
      JNB   _002;
      L     0;
      T     #OUT3;
_002: NOP   0;
NETWORK
TITLE =

      O     #STAT9;
      O     #TEMP13;
      =     #STAT9;
NETWORK
TITLE =

      L     #STAT6;
      L     #IN1;
      >=I   ;
      =     #IO4;
NETWORK
TITLE =

      A     #IO4;
      JCN   M004;
NETWORK
TITLE =

